      IF (_MessageLevel = E_MessageType.eMessageVerbose)
      THEN
        f_MessageSet(_stMsg);
      END_IF

      _rValue                       := Velocity;
    END_IF
END_CASE
CASE _eState
OF
  E_PROGRESS.READY:
    _fbMoveVelocity[2](
                    Axis            := _AxisRef, 
                    Execute         := TRUE,
                    Velocity        := _rValue, 
                    Acceleration    := Acc, 
                    Deceleration    := Dec, 
                    Jerk            := Jerk, 
                    BufferMode      := BufferMode);

    IF _fbMoveVelocity[2].Error
    THEN
      _eState                       := E_PROGRESS.ERROR;

      _nErrorId                     := _fbMoveVelocity[2].ErrorID;
    
      _stMsg.eType                  := E_MessageType.eMessageError;
      _stMsg.eDevice                := e_Device.Axis + TO_DINT(_AxisRef.NcToPlc.AxisId);
      _stMsg.eSubdevice             :=  e_SubDevice.fbMoveVelocity2;
      _stMsg.iErrorNumber           := _nErrorId;

      _stMsg.sText                  := concat(' : ', TO_STRING(_eState));
    
      f_MessageSet(_stMsg);

    ELSIF (_fbMoveVelocity[2].Busy)
    THEN
      _eState                       := E_PROGRESS.PREPARE;

      _stMsg.eType                  := E_MessageType.eMessageVerbose;
      _stMsg.eDevice                := e_Device.Axis + TO_DINT(_AxisRef.NcToPlc.AxisId);
      _stMsg.eSubdevice             :=  e_SubDevice.fbMoveVelocity2;
      _stMsg.iErrorNumber           := 0;

      _stMsg.sText                  := concat('FB busy: ', TO_STRING(_eState));

      IF (_MessageLevel = E_MessageType.eMessageVerbose)
      THEN
        f_MessageSet(_stMsg);
      END_IF

    ELSIF (_fbMoveVelocity[2].CommandAborted)
    THEN
      _eState                       := E_PROGRESS.PREPARE;

      _stMsg.eType                  := E_MessageType.eMessageError;
      _stMsg.eDevice                := e_Device.Axis + TO_DINT(_AxisRef.NcToPlc.AxisId);
      _stMsg.eSubdevice             :=  e_SubDevice.fbMoveVelocity2;
      _stMsg.iErrorNumber           := 0;

      _stMsg.sText                  := concat('FB aborted: ', TO_STRING(_eState));

      f_MessageSet(_stMsg);

    ELSIF (_fbMoveVelocity[2].InVelocity)
    THEN
      _eState                       := E_PROGRESS.PREPARE;

      _stMsg.eType                  := E_MessageType.eMessageVerbose;
      _stMsg.eDevice                := e_Device.Axis + TO_DINT(_AxisRef.NcToPlc.AxisId);
      _stMsg.eSubdevice             :=  e_SubDevice.fbMoveVelocity2;
      _stMsg.iErrorNumber           := 0;

      _stMsg.sText                  := concat('FB done: ', TO_STRING(_eState));

      IF (_MessageLevel = E_MessageType.eMessageVerbose)
      THEN
        f_MessageSet(_stMsg);
      END_IF
    END_IF
END_CASE
CASE _eState
OF
  E_PROGRESS.WAITING:
    _fbMoveVelocity[2](Axis         := _AxisRef);

    IF _fbMoveVelocity[2].Error
    THEN
      _nErrorId                     := _fbMoveVelocity[2].ErrorID;
    
      _stMsg.eType                  := E_MessageType.eMessageError;
      _stMsg.eDevice                := e_Device.Axis + TO_DINT(_AxisRef.NcToPlc.AxisId);
      _stMsg.eSubdevice             :=  e_SubDevice.fbMoveVelocity2;
      _stMsg.iErrorNumber           := _nErrorId;
    
      _stMsg.sText                  := concat(' : ', TO_STRING(_eState));
  
      f_MessageSet(_stMsg);
    
      _eState                       := E_PROGRESS.ERROR;

    ELSIF (Velocity <> _rValue)
    THEN
      _eState                       := E_PROGRESS.STARTUP;

      _fbMoveVelocity[2](
                    Axis            := _AxisRef, 
                    Execute         := FALSE);

      _stMsg.eType                  := E_MessageType.eMessageVerbose;
      _stMsg.eDevice                := e_Device.Axis + TO_DINT(_AxisRef.NcToPlc.AxisId);
      _stMsg.eSubdevice             :=  e_SubDevice.fbMoveVelocity1;
      _stMsg.iErrorNumber           := 0;

      _stMsg.sText                  := concat('Velocity changed: ', TO_STRING(_rValue));
      _stMsg.sText                  := concat(_stMsg.sText        , ' to ');
      _stMsg.sText                  := concat(_stMsg.sText        , TO_STRING(Velocity));

      IF (_MessageLevel = E_MessageType.eMessageVerbose)
      THEN
        f_MessageSet(_stMsg);
      END_IF

      _rValue                       := Velocity;
    END_IF
END_CASE
CASE _eState
OF
  E_PROGRESS.INIT,
  E_PROGRESS.ERROR:
    _fbMoveVelocity[1](Axis         := _AxisRef,
                       Execute      := FALSE);
    _fbMoveVelocity[2](Axis         := _AxisRef,
                       Execute      := FALSE);
END_CASE


MoveVeloBuffer                      := _eState;
END_METHOD

PROPERTY Override : lreal
GET
Override := _rAxisOverride;
END_GET
SET
_rAxisOverride  := Override;
END_SET
END_PROPERTY

METHOD ReadParameter : E_PROGRESS
VAR_INPUT
  Execute           : BOOL;
  ParameterNumber   : Tc2_MC2.MC_AxisParameter;
END_VAR
VAR_INST
  _eState           : E_PROGRESS;
  _rValue           : LREAL;
  _stMsg            : ST_Message;
END_VAR
IF NOT (__ISVALIDREF(_AxisRef)) THEN  ReadParameter  := E_PROGRESS.ERROR; RETURN; END_IF
IF NOT Execute THEN _eState := E_PROGRESS.INIT; END_IF

CASE _eState
OF
  E_PROGRESS.INIT:
    IF Execute 
    THEN
      memset(ADR(_stMsg),0,SIZEOF(_stMsg));
      _nErrorId                     := 0;
      _rValue                       := 0;
      _eState                       := E_PROGRESS.BUSY;
    END_IF
END_CASE
CASE _eState
OF
  E_PROGRESS.BUSY:
    _eState                         := E_PROGRESS.STARTUP;
    _fbReadParameter(
                    Axis            := _AxisRef, 
                    Enable          := FALSE, 
                    ParameterNumber := ParameterNumber, 
                    ReadMode        := Tc2_MC2.READMODE_ONCE, 
                    Value           => _rValue);
END_CASE
CASE _eState
OF
  E_PROGRESS.STARTUP:
    _eState                         := E_PROGRESS.WAITING;
    _fbReadParameter(
                    Axis            := _AxisRef, 
                    Enable          := TRUE, 
                    ParameterNumber := ParameterNumber, 
                    ReadMode        := Tc2_MC2.READMODE_ONCE, 
                    Value           => _rValue);

    _stMsg.eType                    := E_MessageType.eMessageVerbose;
    _stMsg.eDevice                  := e_Device.Axis + TO_DINT(_AxisRef.NcToPlc.AxisId);
    _stMsg.eSubdevice               := e_SubDevice.fbReadParameter;
    _stMsg.iErrorNumber             := 0;

    _stMsg.sText                    := concat(' : ', TO_STRING(_eState));

    IF (_MessageLevel = E_MessageType.eMessageVerbose)
    THEN
      f_MessageSet(_stMsg);
    END_IF
END_CASE
CASE _eState
OF
  E_PROGRESS.WAITING:
    _fbReadParameter(
                    Axis            := _AxisRef,
                    Value           => _rValue);

    IF (_fbReadParameter.Valid)
    THEN
      _eState                       := E_PROGRESS.WORKING;
      _rValueParameterRead          := _rValue;
    ELSE
      IF (_fbReadParameter.Error)
      THEN
        _eState                     := E_PROGRESS.ERROR;
        _nErrorId                   := _fbReadParameter.ErrorID;

        _stMsg.eType                := E_MessageType.eMessageError;
        _stMsg.eDevice              := e_Device.Axis + TO_DINT(_AxisRef.NcToPlc.AxisId);
        _stMsg.eSubdevice           := e_SubDevice.fbReadParameter;
        _stMsg.iErrorNumber         := _nErrorId;

        _stMsg.sText                := concat(' : ', TO_STRING(_eState));

        f_MessageSet(_stMsg);

        _fbReadParameter(
                    Axis            := _AxisRef, 
                    Enable          := FALSE);
      END_IF
    END_IF
END_CASE
CASE _eState
OF
  E_PROGRESS.WORKING:
    _eState                         := E_PROGRESS.DONE;
    _fbReadParameter(
                    Axis            := _AxisRef, 
                    Enable          := FALSE);

    _stMsg.eType                    := E_MessageType.eMessageVerbose;
    _stMsg.eDevice                  := e_Device.Axis + TO_DINT(_AxisRef.NcToPlc.AxisId);
    _stMsg.eSubdevice               := e_SubDevice.fbReadParameter;
    _stMsg.iErrorNumber             := 0;

    _stMsg.sText                    := concat(' : ', TO_STRING(_eState));

    IF (_MessageLevel = E_MessageType.eMessageVerbose)
    THEN
      f_MessageSet(_stMsg);
    END_IF
END_CASE

ReadParameter                       := _eState;
END_METHOD

PROPERTY ReadParameterValue : LREAL
GET
ReadParameterValue := _rValueParameterRead;
END_GET
END_PROPERTY

METHOD Reset : E_PROGRESS
VAR_INPUT
  Execute           : BOOL;
END_VAR
VAR_INST
  _eState           : E_PROGRESS;
  _rValue           : LREAL;
  _stMsg            : ST_Message;
END_VAR
IF NOT (__ISVALIDREF(_AxisRef)) THEN  Reset  := E_PROGRESS.ERROR; RETURN; END_IF
IF NOT Execute THEN _eState := E_PROGRESS.INIT; END_IF

CASE _eState
OF
  E_PROGRESS.INIT:
    IF Execute 
    THEN
      memset(ADR(_stMsg),0,SIZEOF(_stMsg));
      _nErrorId                   := 0;
      _rValue                     := 0;
      _eState                     := E_PROGRESS.BUSY;
    END_IF
END_CASE
CASE _eState
OF
  E_PROGRESS.BUSY:
    _eState                       := E_PROGRESS.WAITING;
    _fbReset(
              Axis                := _AxisRef, 
              Execute             := FALSE);
END_CASE
CASE _eState
OF
  E_PROGRESS.WAITING:
    _fbReset(
              Axis                := _AxisRef, 
              Execute             := TRUE);

    _AxisRef();

    IF _fbReset.Error
    THEN
      _nErrorId                   := _fbReset.ErrorID;

      _stMsg.eType                := E_MessageType.eMessageError;
      _stMsg.eDevice              := e_Device.Axis + TO_DINT(_AxisRef.NcToPlc.AxisId);
      _stMsg.eSubdevice           := e_SubDevice.fbReset;
      _stMsg.iErrorNumber         := _nErrorId;

      f_MessageSet(_stMsg);
      _fbReset(
              Axis                := _AxisRef, 
              Execute             := FALSE);

      _eState                     := E_PROGRESS.ERROR;
    ELSE
      IF _fbReset.Done OR NOT
         _fbReset.Busy
      THEN
        _eState                   := E_PROGRESS.WORKING;
      END_IF
    END_IF
END_CASE
CASE _eState
OF
  E_PROGRESS.WORKING:
    _eState                       := E_PROGRESS.DONE;
    _fbReset(
              Axis                := _AxisRef, 
              Execute             := FALSE);

    _stMsg.eType                  := E_MessageType.eMessageVerbose;
    _stMsg.eDevice                := e_Device.Axis + TO_DINT(_AxisRef.NcToPlc.AxisId);
    _stMsg.eSubdevice             := e_SubDevice.fbReset;
    _stMsg.iErrorNumber           := 0;

    _stMsg.sText                    := concat(' : ', TO_STRING(_eState));

    IF (_MessageLevel = E_MessageType.eMessageVerbose)
    THEN
      f_MessageSet(_stMsg);
    END_IF
END_CASE


Reset                             := _eState;
END_METHOD

METHOD SendToPos : E_PROGRESS
VAR_INPUT
  Execute         : BOOL;
  Position        : LREAL;
  Vel             : LREAL;
  Acc             : LREAL;
  Dec             : LREAL;
  Jerk            : LREAL;
  BufferMode      : Tc2_MC2.MC_BufferMode;
END_VAR
VAR_INST
  _eState           : E_PROGRESS;
  _rValue           : LREAL;
  _rTarget          : LREAL := 0.5;
  _stMsg            : ST_Message;
END_VAR
IF NOT (__ISVALIDREF(_AxisRef)) THEN  SendToPos  := E_PROGRESS.ERROR; RETURN; END_IF
IF NOT Execute THEN _eState := E_PROGRESS.INIT; END_IF

CASE _eState
OF
  E_PROGRESS.INIT:
    IF Execute 
    THEN
      memset(ADR(_stMsg),0,SIZEOF(_stMsg));
      _nErrorId                     := 0;
      _rValue                       := 0;
      _eState                       := E_PROGRESS.BUSY;

      _stMsg.eType                  := E_MessageType.eMessageVerbose;
      _stMsg.eDevice                := e_Device.Axis + TO_DINT(_AxisRef.NcToPlc.AxisId);
      _stMsg.eSubdevice             := e_SubDevice.fbMoveAbsolute1;
      _stMsg.iErrorNumber           := 0;

      _stMsg.sText                  := concat(' : ', TO_STRING(Position));

      IF (_MessageLevel = E_MessageType.eMessageVerbose)
      THEN
        f_MessageSet(_stMsg);
      END_IF
    END_IF
END_CASE
CASE _eState
OF
  E_PROGRESS.BUSY:
    _eState                         := E_PROGRESS.STARTUP;
    _rValue                         := Position;

    _fbMoveAbsolute[1](Axis         := _AxisRef,
                       Execute      := FALSE);
END_CASE
CASE _eState
OF
  E_PROGRESS.STARTUP:
    _fbMoveAbsolute[1](
                    Axis            := _AxisRef, 
                    Execute         := TRUE,
                    Position        := _rValue, 
                    Velocity        := Vel, 
                    Acceleration    := Acc, 
                    Deceleration    := Dec, 
                    Jerk            := Jerk, 
                    BufferMode      := BufferMode);

    _eState                         := E_PROGRESS.PREPARE;
END_CASE
CASE _eState
OF
  E_PROGRESS.PREPARE:
    _fbMoveAbsolute[1](Axis         := _AxisRef);

    IF (_fbMoveAbsolute[1].Error)
    THEN
      _nErrorId                     := _fbMoveAbsolute[1].ErrorID;
    
      _stMsg.eType                  := E_MessageType.eMessageError;
      _stMsg.eDevice                := e_Device.Axis + TO_DINT(_AxisRef.NcToPlc.AxisId);
      _stMsg.eSubdevice             :=  e_SubDevice.fbMoveAbsolute1;
      _stMsg.iErrorNumber           := _nErrorId;
    
      f_MessageSet(_stMsg);
    
      _eState                         := E_PROGRESS.ERROR;

    ELSIF (_fbMoveAbsolute[1].Active)
    THEN
      _eState                       := E_PROGRESS.WAITING;
    END_IF
END_CASE
CASE _eState
OF
  E_PROGRESS.WAITING:
    _fbMoveAbsolute[1](Axis         := _AxisRef);

    IF (_fbMoveAbsolute[1].Error)
    THEN
      _nErrorId                     := _fbMoveAbsolute[1].ErrorID;
    
      _stMsg.eType                  := E_MessageType.eMessageError;
      _stMsg.eDevice                := e_Device.Axis + TO_DINT(_AxisRef.NcToPlc.AxisId);
      _stMsg.eSubdevice             :=  e_SubDevice.fbMoveAbsolute1;
      _stMsg.iErrorNumber           := _nErrorId;
    
      f_MessageSet(_stMsg);
    
      _eState                         := E_PROGRESS.ERROR;

    ELSIF (_AxisRef.NcToPlc.ActPos > _fbMoveAbsolute[1].Position + _rTarget)
    THEN
      _fbMoveAbsolute[1](Axis       := _AxisRef,
                         Execute    := FALSE);

      _eState                       := E_PROGRESS.DONE;

      _stMsg.eType                  := E_MessageType.eMessageVerbose;
      _stMsg.eDevice                := e_Device.Axis + TO_DINT(_AxisRef.NcToPlc.AxisId);
      _stMsg.eSubdevice             := e_SubDevice.fbMoveAbsolute1;
      _stMsg.iErrorNumber           := 0;

      _stMsg.sText                  := concat(' : ', TO_STRING(_eState));

      IF (_MessageLevel = E_MessageType.eMessageVerbose)
      THEN
        f_MessageSet(_stMsg);
      END_IF
    END_IF
END_CASE

SendToPos                             := _eState;
END_METHOD

METHOD StartUp : E_PROGRESS
VAR_INPUT
  Execute           : BOOL;
END_VAR
VAR_INST
  _eState           : E_PROGRESS;
  _uiEncType        : UDINT;

  _sEncoder,
  _sName            : STRING(30);

  _rValue           : LREAL;
  _stMsg            : ST_Message;
END_VAR
IF NOT (__ISVALIDREF(_AxisRef)) THEN  StartUp  := E_PROGRESS.ERROR; RETURN; END_IF
IF NOT Execute THEN _eState := E_PROGRESS.INIT; END_IF


CASE _eState
OF
  E_PROGRESS.INIT:
    IF Execute 
    THEN
      memset(ADR(_stMsg),0,SIZEOF(_stMsg));
      _nErrorId                     := 0;
      _rValue                       := 0;
      _eState                       := E_PROGRESS.BUSY;
    END_IF
END_CASE
CASE _eState
OF
  E_PROGRESS.BUSY:
    IF (_AxisRef.NcToPlc.AxisId <> 0)
    THEN
      _stMsg.eType                  := E_MessageType.eMessageVerbose;
      _stMsg.eDevice                := e_Device.Axis + TO_DINT(_AxisRef.NcToPlc.AxisId);
      _stMsg.eSubdevice             := e_Subdevice.AxisStartUp;
      _stMsg.iErrorNumber           := 0;
      _stMsg.sText                  := concat('StartUp NcAxisId: ', TO_STRING(_AxisRef.NcToPlc.AxisId));

      IF (_MessageLevel = E_MessageType.eMessageVerbose)
      THEN
        f_MessageSet(_stMsg);
      END_IF

      _eState                       := E_PROGRESS.STARTUP;
    END_IF
END_CASE
CASE _eState
OF
  E_PROGRESS.STARTUP:
    _fbADSRead(
              NETID                 := '', 
              PORT                  := 501, 
              IDXGRP                := (16#5000 + _AxisRef.NcToPlc.AxisId), 
              IDXOFFS               := 16#00000003, // offset for encoder type
              LEN                   := SIZEOF(_nEncoderType), 
              DESTADDR              := ADR(_nEncoderType),
              TMOUT                 := T#200MS,
              READ                  := FALSE);

    // clear required ADS information
    _sAxisName      := _sName       := 'NO NAME';
    _sEncoderType   := _sEncoder    := 'NO TYPE';
    _nEncoderType   := _uiEncType   :=  0;

    _eState                         := E_PROGRESS.PREPARE;
END_CASE
CASE _eState
OF
  E_PROGRESS.PREPARE:
    _fbADSRead(
              NETID                 := '', 
              PORT                  := 501, 
              IDXGRP                := (16#5000 + _AxisRef.NcToPlc.AxisId), 
              IDXOFFS               := 16#00000003, // offset for encoder type
              LEN                   := SIZEOF(_nEncoderType), 
              DESTADDR              := ADR(_nEncoderType),
              TMOUT                 := T#200MS,
              READ                  := TRUE);

    IF (_fbADSRead.ERR)
    THEN
      _nErrorId                     := _fbAdsRead.ERRID;

      _stMsg.eType                  := E_MessageType.eMessageError;
      _stMsg.eDevice                := e_Device.Axis + TO_DINT(_AxisRef.NcToPlc.AxisId);
      _stMsg.eSubdevice             := e_Subdevice.AxisStartUp;
      _stMsg.iErrorNumber           := _nErrorId;
      _stMsg.sText                  := 'StartUp Ads Error Read Encoder Type';

      f_MessageSet(_stMsg);
      _eState                       := E_PROGRESS.ERROR;

    ELSIF (_nEncoderType <> 0)
    THEN
      _uiEncType  := _eEncoderType  := _nEncoderType;
      _sEncoder   := _sEncoderType  := TO_STRING(_eEncoderType);

      _stMsg.eType                  := E_MessageType.eMessageInfo;
      _stMsg.eDevice                := e_Device.Axis + TO_DINT(_AxisRef.NcToPlc.AxisId);
      _stMsg.eSubdevice             := e_Subdevice.AxisStartUp;
      _stMsg.iErrorNumber           := 0;
      _stMsg.sText                  := concat('Encoder Type: ', _sEncoder);

      IF (_MessageLevel < E_MessageType.eMessageError)
      THEN
        f_MessageSet(_stMsg);
      END_IF

      _eState                       := E_PROGRESS.READY;
    END_IF
END_CASE
CASE _eState
OF
  E_PROGRESS.READY:
    _fbADSRead(
            NETID                   := '', 
            PORT                    := 501, 
            IDXGRP                  := (16#4000 + _AxisRef.NcToPlc.AxisId), 
            IDXOFFS                 := 16#00000002, // offset for axis name
            LEN                     := SIZEOF(_sAxisName), 
            DESTADDR                := ADR(_sAxisName),
            READ                    := FALSE);

    _eState                         := E_PROGRESS.WAITING;
END_CASE
CASE _eState
OF
  E_PROGRESS.WAITING:
    _fbADSRead(
            NETID                   := '', 
            PORT                    := 501, 
            IDXGRP                  := (16#4000 + _AxisRef.NcToPlc.AxisId), 
            IDXOFFS                 := 16#00000002, // offset for axis name
            LEN                     := SIZEOF(_sAxisName), 
            DESTADDR                := ADR(_sAxisName),
            READ                    := TRUE);

    IF (_fbADSRead.ERR)
    THEN
      _nErrorId                     := _fbAdsRead.ERRID;

      _stMsg.eType                  := E_MessageType.eMessageError;
      _stMsg.eDevice                := e_Device.Axis + TO_DINT(_AxisRef.NcToPlc.AxisId);;
      _stMsg.eSubdevice             := e_Subdevice.AxisStartUp;
      _stMsg.iErrorNumber           := _nErrorId;
      _stMsg.sText                  := 'StartUp Ads Error Read Axis Name';

      f_MessageSet(_stMsg);
      _eState                       := E_PROGRESS.ERROR;

    ELSIF (_sAxisName <> 'NO NAME')
    THEN
      _sName                        := _sAxisName;

      _stMsg.eType                  := E_MessageType.eMessageInfo;
      _stMsg.eDevice                := e_Device.Axis + TO_DINT(_AxisRef.NcToPlc.AxisId);;
      _stMsg.eSubdevice             := e_Subdevice.AxisStartUp;
      _stMsg.iErrorNumber           := 0;
      _stMsg.sText                  := concat('Axis Name: ', _sName);

      IF (_MessageLevel < E_MessageType.eMessageError)
      THEN
        f_MessageSet(_stMsg);
      END_IF

      _eState                       := E_PROGRESS.WORKING;
    END_IF
END_CASE
CASE _eState
OF
  E_PROGRESS.WORKING:
    _eState                         := E_PROGRESS.DONE;
END_CASE

StartUp                             := _eState;
END_METHOD

METHOD Stop : E_PROGRESS
VAR_INPUT
  Execute           : BOOL;
  Dec               : LREAL;
  Jerk              : LREAL;

END_VAR
VAR_INST
  _eState           : E_PROGRESS;
  _rValue           : LREAL;
  _stMsg            : ST_Message;
END_VAR
IF NOT (__ISVALIDREF(_AxisRef)) THEN  Stop  := E_PROGRESS.ERROR; RETURN; END_IF
IF NOT Execute THEN _eState := E_PROGRESS.INIT; END_IF

CASE _eState
OF
  E_PROGRESS.INIT:
    IF Execute 
    THEN
      memset(ADR(_stMsg),0,SIZEOF(_stMsg));
      _nErrorId                     := 0;
      _rValue                       := 0;
      _eState                       := E_PROGRESS.BUSY;
    END_IF
END_CASE
CASE _eState
OF
  E_PROGRESS.BUSY:
    _eState                         := E_PROGRESS.WAITING;
    _fbStop(
              Axis                  := _AxisRef, 
              Execute               := FALSE, 
              Deceleration          := Dec, 
              Jerk                  := Jerk);
END_CASE
CASE _eState
OF
  E_PROGRESS.WAITING:
    _fbStop(
              Axis                  := _AxisRef, 
              Execute               := TRUE, 
              Deceleration          := Dec, 
              Jerk                  := Jerk);

    IF _fbStop.Error
    THEN
        _nErrorId                   := _fbStop.ErrorID;

        _stMsg.eType                := E_MessageType.eMessageError;
        _stMsg.eDevice              := e_Device.Axis + TO_DINT(_AxisRef.NcToPlc.AxisId);
        _stMsg.eSubdevice           := e_SubDevice.fbStop;
        _stMsg.iErrorNumber         := _nErrorId;

        f_MessageSet(_stMsg);
        _fbStop(
              Axis                  := _AxisRef, 
              Execute               := FALSE);

      _eState                       := E_PROGRESS.ERROR;

    ELSE
      IF _fbStop.Done OR
         _AxisRef.Status.NotMoving
      THEN
        _eState                     := E_PROGRESS.WORKING;

      ELSIF _fbStop.CommandAborted
      THEN
        _eState                     := E_PROGRESS.BUSY;
      END_IF
    END_IF
END_CASE
CASE _eState
OF
  E_PROGRESS.WORKING:
    _fbStop(
              Axis                  := _AxisRef, 
              Execute               := FALSE);

    _eState                         := E_PROGRESS.DONE;
END_CASE


Stop                                := _eState;
END_METHOD

METHOD Template : E_PROGRESS
VAR_INPUT
  Execute           : BOOL;
END_VAR
VAR_INST
  _eState           : E_PROGRESS;
  _rValue           : LREAL;
  _udiErr           : UDINT;
  _stMsg            : ST_Message;


END_VAR
IF NOT (__ISVALIDREF(_AxisRef)) THEN _eState := E_PROGRESS.ERROR; END_IF
IF NOT Execute THEN _eState := E_PROGRESS.INIT; END_IF

CASE _eState
OF
  E_PROGRESS.INIT:
    IF Execute 
    THEN
      memset(ADR(_stMsg),0,SIZEOF(_stMsg));
      _udiErr                       := 0;
      _rValue                       := 0;
      _eState                       := E_PROGRESS.BUSY;
    END_IF
END_CASE
CASE _eState
OF
  E_PROGRESS.BUSY:
    _eState                         := E_PROGRESS.STARTUP;
END_CASE
CASE _eState
OF
  E_PROGRESS.STARTUP:
    _eState                       := E_PROGRESS.PREPARE;
END_CASE
CASE _eState
OF
  E_PROGRESS.PREPARE:
    _eState                         := E_PROGRESS.READY;
END_CASE
CASE _eState
OF
  E_PROGRESS.READY:
    _eState                         := E_PROGRESS.WAITING;
END_CASE
CASE _eState
OF
  E_PROGRESS.WAITING:
    _eState                         := E_PROGRESS.WORKING;
END_CASE
CASE _eState
OF
  E_PROGRESS.WORKING:
    _eState                         := E_PROGRESS.DONE;
END_CASE

Template_1 := _eState;
END_METHOD

METHOD WriteParameter : E_PROGRESS
VAR_INPUT
  Execute           : BOOL;
  Value             : LREAL;
  ParameterNumber   : Tc2_MC2.MC_AxisParameter;
END_VAR
VAR_INST
  _eState           : E_PROGRESS;
  _nParameter       : Tc2_MC2.MC_AxisParameter;
  _rValue           : LREAL;
  _stMsg            : ST_Message;
END_VAR
IF NOT (__ISVALIDREF(_AxisRef)) THEN  WriteParameter  := E_PROGRESS.ERROR; RETURN; END_IF
IF NOT Execute THEN _eState := E_PROGRESS.INIT; END_IF

CASE _eState
OF
  E_PROGRESS.INIT:
    IF Execute 
    THEN
      memset(ADR(_stMsg),0,SIZEOF(_stMsg));
      _nParameter                   := 0;
      _nErrorId                     := 0;
      _rValue                       := 0;
      _eState                       := E_PROGRESS.BUSY;
    END_IF
END_CASE
CASE _eState
OF
  E_PROGRESS.BUSY:
    _eState                         := E_PROGRESS.STARTUP;
    _nParameter                     := ParameterNumber;

    _fbWriteParameter(
                    Axis            := _AxisRef, 
                    Execute         := FALSE, 
                    ParameterNumber := ParameterNumber, 
                    Value           := Value);
END_CASE
CASE _eState
OF
  E_PROGRESS.STARTUP:
    _eState                         := E_PROGRESS.WAITING;
    _fbWriteParameter(
                    Axis            := _AxisRef, 
                    Execute         := TRUE, 
                    ParameterNumber := ParameterNumber, 
                    Value           := Value);

END_CASE
CASE _eState
OF
  E_PROGRESS.WAITING:
    _fbWriteParameter(
                    Axis            := _AxisRef, 
                    ParameterNumber := ParameterNumber, 
                    Value           := Value);

    IF _fbWriteParameter.Error
    THEN
      _nErrorId                     := _fbWriteParameter.ErrorID;

      _stMsg.eType                  := E_MessageType.eMessageError;
      _stMsg.eDevice                := e_Device.Axis + TO_DINT(_AxisRef.NcToPlc.AxisId);
      _stMsg.eSubdevice             := e_SubDevice.fbWriteParameter;
      _stMsg.iErrorNumber           := _nErrorId;

      f_MessageSet(_stMsg);

      _fbWriteParameter(
                    Axis            := _AxisRef,
                    Execute         := FALSE, 
                    ParameterNumber := ParameterNumber, 
                    Value           := Value);


      _eState                       := E_PROGRESS.ERROR;
    ELSE
      IF _fbWriteParameter.Done
      THEN
        _rValue                     := _fbWriteParameter.Value;
        _eState                     := E_PROGRESS.WORKING;
      END_IF
    END_IF

END_CASE
CASE _eState
OF
  E_PROGRESS.WORKING:
    _fbWriteParameter(
                    Axis            := _AxisRef,
                    Execute         := FALSE, 
                    ParameterNumber := ParameterNumber, 
                    Value           := Value);
    _eState                         := E_PROGRESS.DONE;
END_CASE


WriteParameter                      := _eState;
END_METHOD

METHOD WriteParameterPersistent : E_PROGRESS
VAR_INPUT
  Execute           : BOOL;
  Value             : LREAL;
  ParameterNumber   : Tc2_MC2.MC_AxisParameter;
END_VAR
VAR_INST
  _eState           : E_PROGRESS;
  _rValue           : LREAL;
  _stMsg            : ST_Message;
END_VAR
IF NOT (__ISVALIDREF(_AxisRef)) THEN  WriteParameterPersistent  := E_PROGRESS.ERROR; RETURN; END_IF
IF NOT Execute THEN _eState := E_PROGRESS.INIT; END_IF

CASE _eState
OF
  E_PROGRESS.INIT:
    IF Execute 
    THEN
      memset(ADR(_stMsg),0,SIZEOF(_stMsg));
      _nErrorId                     := 0;
      _rValue                       := 0;
      _eState                       := E_PROGRESS.BUSY;
    END_IF
END_CASE
CASE _eState
OF
  E_PROGRESS.BUSY:
    _eState                         := E_PROGRESS.STARTUP;
    _fbWriteParameterPersist(
                    Axis            := _AxisRef, 
                    Execute         := FALSE, 
                    ParameterNumber := ParameterNumber, 
                    Value           := Value);
END_CASE
CASE _eState
OF
  E_PROGRESS.STARTUP:
    _eState                         := E_PROGRESS.WAITING;
    _fbWriteParameterPersist(
                    Axis            := _AxisRef, 
                    Execute         := TRUE, 
                    ParameterNumber := ParameterNumber, 
                    Value           := Value);

END_CASE
CASE _eState
OF
  E_PROGRESS.WAITING:
    _fbWriteParameterPersist(
                    Axis            := _AxisRef, 
                    ParameterNumber := ParameterNumber, 
                    Value           := Value);

    IF (_fbWriteParameterPersist.Error)
    THEN
      _nErrorId                     := _fbWriteParameterPersist.ErrorID;

      _stMsg.eType                  := E_MessageType.eMessageError;
      _stMsg.eDevice                := e_Device.Axis + TO_DINT(_AxisRef.NcToPlc.AxisId);
      _stMsg.eSubdevice             := e_SubDevice.fbWriteParameterPersistent;
      _stMsg.iErrorNumber           := _nErrorId;

      f_MessageSet(_stMsg);

      _fbWriteParameterPersist(
                    Axis            := _AxisRef,
                    Execute         := FALSE, 
                    ParameterNumber := ParameterNumber, 
                    Value           := Value);


      _eState                       := E_PROGRESS.ERROR;
    ELSE
      IF (_fbWriteParameterPersist.Done)
      THEN
        _rValue                     := _fbWriteParameterPersist.Value;
        _eState                     := E_PROGRESS.WORKING;
      END_IF
    END_IF

END_CASE
CASE _eState
OF
  E_PROGRESS.WORKING:
    _fbWriteParameterPersist(
                    Axis            := _AxisRef,
                    Execute         := FALSE, 
                    ParameterNumber := ParameterNumber, 
                    Value           := Value);

    _eState                         := E_PROGRESS.DONE;
END_CASE


WriteParameterPersistent            := _eState;
END_METHOD

END_FUNCTION_BLOCK

// ---- CAM/FB_CamCtrl.TcPOU
FUNCTION_BLOCK FB_CamCtrl EXTENDS FB_CamAxis IMPLEMENTS I_Cam_Ctrl
VAR
  _eInit                    : E_PROGRESS;
  _nAxisIndex               : UINT;       // know thyself

  // get interface from McAxis for access to Reset, Enable, Disable, Halt
  _ItfMcAxis                : ARRAY[1..PLC_CONSTANT.MAX_AXIS] OF I_McAxis;

  // pointers to all; access required for coupling; access by index
  _Axes                     : REFERENCE TO ARRAY[1..PLC_CONSTANT.MAX_AXIS] OF AXIS_REF;

  _Ctrl                     : POINTER TO ARRAY[1..PLC_CONSTANT.MAX_AXIS] OF ST_CAM_CTRL;    // contains command to be executed
  _State                    : POINTER TO ARRAY[1..PLC_CONSTANT.MAX_AXIS] OF ST_CAM_STATE;   // mirrors command with added result

  _Info                     : POINTER TO ARRAY[1..PLC_CONSTANT.MAX_AXIS] OF ST_CAM_INFO;    // Read Camming Info Data
  _Data                     : POINTER TO ARRAY[1..PLC_CONSTANT.MAX_AXIS] OF ST_CAM_DATA;    // Camming parameters

  _MotionFunction           : POINTER TO ARRAY[1..PLC_CONSTANT.MAX_AXIS] OF ST_MOTION_FUNCTION;
  _MotionFunctionPoint      : POINTER TO ARRAY[1..PLC_CONSTANT.MAX_AXIS] OF ST_MOTION_FUNCTION_POINT;

  // local copies of command
  _eCtrl,
  _eCtrlOld                       : E_AXIS_CTRL;

  // execution state
  _eResult                        : E_PROGRESS;   // result of execution state
  _eResultOld                     : E_PROGRESS;   // old result for detecting change
  _eState                         : E_AXIS_STATE; // execution state
END_VAR

PROPERTY Axes : reference TO ARRAY[1..PLC_CONSTANT.MAX_AXIS] OF AXIS_REF
SET
_Axes := Axes;
END_SET
END_PROPERTY

METHOD AxisCamIdle : E_PROGRESS
VAR_INPUT
  Execute           : BOOL;
END_VAR
VAR_INST
  _eResult,
  _eState           : E_PROGRESS;
  _stMsg            : ST_Message;
  _nRetry           : UINT;
END_VAR
IF NOT Execute THEN _eState := E_PROGRESS.INIT; END_IF
IF NOT Check() THEN _eState := E_PROGRESS.ERROR; END_IF

CASE _eState
OF
  E_PROGRESS.INIT:
    IF Execute 
    THEN
      memset(ADR(_stMsg),0,SIZEOF(_stMsg));
      _nRetry                       := 0;
      _eResult                      := _ItfMcAxis[_nAxisIndex].Reset(FALSE);
      _eState                       := E_PROGRESS.BUSY;
    END_IF
END_CASE
CASE _eState
OF
  E_PROGRESS.PREPARE:
    _nRetry                         := _nRetry + 1;
    _eResult                        := _ItfMcAxis[_nAxisIndex].Reset(FALSE);
    _eResult                        := _ItfMcAxis[_nAxisIndex].Enable(FALSE);

    _eState                         := E_PROGRESS.BUSY;

    _stMsg.eType                    := E_MessageType.eMessageInfo;
    _stMsg.eDevice                  := e_Device.Camming + TO_DINT(_AxisSlave.NcToPlc.AxisId);
    _stMsg.eSubdevice               :=  e_SubDevice.fbPowerOn;
    _stMsg.iErrorNumber             := _nErrorId;

    _stMsg.sText                    := concat(TO_STRING(_eCtrl), ' retry: ');
    _stMsg.sText                    := concat(_stMsg.sText, TO_STRING(_nRetry));

    IF (_MessageLevel < E_MessageType.eMessageError)
    THEN
      f_MessageSet(_stMsg);
    END_IF
END_CASE
CASE _eState
OF
  E_PROGRESS.BUSY:
    _eResult                        := _ItfMcAxis[_nAxisIndex].Reset(TRUE);

    IF (_eResult = E_PROGRESS.DONE)
    THEN
      _eState                       := E_PROGRESS.STARTUP;
    END_IF
END_CASE
CASE _eState
OF
  E_PROGRESS.STARTUP:
    _eResult                        := _ItfMcAxis[_nAxisIndex].Reset(FALSE);
    _eResult                        := _ItfMcAxis[_nAxisIndex].Enable(FALSE);
    _eState                         := E_PROGRESS.READY;
END_CASE
CASE _eState
OF
  E_PROGRESS.READY:
    _eResult                        := _ItfMcAxis[_nAxisIndex].Enable(TRUE);

    IF (_nRetry > MAX_RETRY)
    THEN
      _eState                       := E_PROGRESS.ERROR;

    ELSIF (_eResult = E_PROGRESS.DONE)
    THEN
      _ItfMcAxis[_nAxisIndex].Enable(FALSE);
      _eState                       := E_PROGRESS.DONE;

    ELSIF (_eResult = E_PROGRESS.ERROR)
    THEN
      _eState                       := E_PROGRESS.PREPARE;

      _nErrorId                     := _AxisSlave.NcToPlc.ErrorCode;
    
      _stMsg.eType                  := E_MessageType.eMessageError;
      _stMsg.eDevice                := e_Device.Camming + TO_DINT(_AxisSlave.NcToPlc.AxisId);
      _stMsg.eSubdevice             :=  e_SubDevice.fbPowerOn;
      _stMsg.iErrorNumber           := _nErrorId;

      _stMsg.sText                  := concat(TO_STRING(_eCtrl), ' error axis enable: ');
      _stMsg.sText                  := concat(_stMsg.sText, TO_STRING(_nAxisIndex));

      f_MessageSet(_stMsg);
    END_IF
END_CASE

AxisCamIdle                                := _eState;
END_METHOD

METHOD AxisCamIn : E_PROGRESS
VAR_INPUT
  Execute           : BOOL;
END_VAR
VAR_INST
  _eCk              : E_CHECK_STATE;

  _eResult,
  _eState           : E_PROGRESS;
  _rValue           : LREAL;
  _udiErr           : UDINT;
  _stMsg            : ST_Message;

END_VAR
IF NOT Execute THEN _eState := E_PROGRESS.INIT; END_IF
IF NOT Check() THEN _eState := E_PROGRESS.ERROR; END_IF


CASE _eState
OF
  E_PROGRESS.INIT:
    IF Execute 
    THEN
      memset(ADR(_stMsg),0,SIZEOF(_stMsg));
      _udiErr                       := 0;

      IF NOT (_stCamData.nMasterIndex > 0) OR
         NOT (_stCamData.nMasterIndex < PLC_CONSTANT.MAX_AXIS+1)
      THEN
        _eState                     := E_PROGRESS.ERROR;
        _eCk                        := E_CHECK_STATE.CAM_MASTER_AXIS_REF_INVALID;

        _stMsg.eType                := E_MessageType.eMessageError;
        _stMsg.eDevice              := E_Device.Camming + TO_DINT(_AxisSlave.NcToPlc.AxisId);
        _stMsg.eSubdevice           := e_Subdevice.CamControl;
        _stMsg.iErrorNumber         := _stCamData.nMasterIndex;
  
        _stMsg.sText                := concat(' : ', TO_STRING(_eCk));
        f_MessageSet(_stMsg);

      ELSE
        _eState                     := E_PROGRESS.BUSY;
        _eCk                        := E_CHECK_STATE.CHECK_DONE;
        _eResult                    := CamIn(FALSE, _stCamData.nMasterIndex);
      END_IF
    END_IF
END_CASE
CASE _eState
OF
  E_PROGRESS.BUSY:
      _eResult                      := CamIn(TRUE, _stCamData.nMasterIndex);

    IF (_eResult = E_PROGRESS.ERROR)
    THEN
      CamIn(FALSE, _stCamData.nMasterIndex);
      _eState                       := E_PROGRESS.ERROR;
      _udiErr                       := _fbCamInV2.ErrorID;

    ELSIF (_eResult = E_PROGRESS.DONE)
    THEN
      CamIn(FALSE, _stCamData.nMasterIndex);
      _eState                       := E_PROGRESS.DONE;
    END_IF
END_CASE


AxisCamIn                           := _eState;
END_METHOD

METHOD AxisCamInfo : E_PROGRESS
VAR_INPUT
  Execute           : BOOL;
END_VAR
VAR_INST
  _eCk              : E_CHECK_STATE;

  _eResult,
  _eState           : E_PROGRESS;
  _rValue           : LREAL;
  _udiErr           : UDINT;
  _stMsg            : ST_Message;

END_VAR
IF NOT Execute THEN _eState := E_PROGRESS.INIT; END_IF
IF NOT Check() THEN _eState := E_PROGRESS.ERROR; END_IF


CASE _eState
OF
  E_PROGRESS.INIT:
    IF Execute 
    THEN
      memset(ADR(_stMsg),0,SIZEOF(_stMsg));
      _udiErr                       := 0;

      _eState                       := E_PROGRESS.BUSY;
      _eCk                          := E_CHECK_STATE.CHECK_DONE;
      _eResult                      := CamInfo(FALSE, _stCamData.nCamTableId, _stCamData.bAtMasterPosition, _stCamData.rMasterPosition);
    END_IF
END_CASE
CASE _eState
OF
  E_PROGRESS.BUSY:
      _eResult                      := CamInfo(TRUE, _stCamData.nCamTableId, _stCamData.bAtMasterPosition, _stCamData.rMasterPosition);

    IF (_eResult = E_PROGRESS.ERROR)
    THEN
      _eState                       := E_PROGRESS.ERROR;
      CamInfo(FALSE, _stCamData.nCamTableId, _stCamData.bAtMasterPosition, _stCamData.rMasterPosition);

    ELSIF (_eResult = E_PROGRESS.DONE)
    THEN
      _eState                       := E_PROGRESS.READY;
      CamInfo(FALSE, _stCamData.nCamTableId, _stCamData.bAtMasterPosition, _stCamData.rMasterPosition);
    END_IF
END_CASE
CASE _eState
OF
  E_PROGRESS.READY:
    _Info^[_nAxisIndex]             := CamInfoData;

    _stMsg.eType                    := E_MessageType.eMessageInfo;
    _stMsg.eDevice                  := E_Device.Camming + TO_DINT(_AxisSlave.NcToPlc.AxisId);
    _stMsg.eSubdevice               := e_Subdevice.CamControl;
    _stMsg.iErrorNumber             := 0;

    _stMsg.sText                    := concat('CamInfoData : ', TO_STRING(_eState));

    IF (_MessageLevel < E_MessageType.eMessageError)
    THEN
      f_MessageSet(_stMsg);
    END_IF

    _eState                         := E_PROGRESS.DONE;
END_CASE


AxisCamInfo                         := _eState;
END_METHOD

METHOD AxisCamOut : E_PROGRESS
VAR_INPUT
  Execute           : BOOL;
END_VAR
VAR_INST
  _eResult,
  _eState           : E_PROGRESS;
END_VAR
IF NOT Execute THEN _eState := E_PROGRESS.INIT; END_IF
IF NOT Check() THEN _eState := E_PROGRESS.ERROR; END_IF


CASE _eState
OF
  E_PROGRESS.INIT:
    IF Execute 
    THEN
      _eState                       := E_PROGRESS.BUSY;
      _eResult                      := CamOut(FALSE);
    END_IF
END_CASE
CASE _eState
OF
  E_PROGRESS.BUSY:
    _eResult                        := CamOut(TRUE);

    IF (_eResult = E_PROGRESS.ERROR)
    THEN
      CamOut(FALSE);
      _eState                       := E_PROGRESS.ERROR;

    ELSIF (_eResult = E_PROGRESS.DONE)
    THEN
      CamOut(FALSE);
      _eState                       := E_PROGRESS.DONE;
    END_IF
END_CASE


AxisCamOut                          := _eState;
END_METHOD

METHOD AxisCamScaling : E_PROGRESS
VAR_INPUT
  Execute             : BOOL;
END_VAR
VAR_INST
  _eResult,
  _eState             : E_PROGRESS;
  _rValue             : LREAL;
  _udiErr             : UDINT;
  _stMsg              : ST_Message;
END_VAR

IF NOT __ISVALIDREF(_AxisSlave)
THEN
  _eCheck                   := E_CHECK_STATE.CAM_SLAVE_AXIS_REF_INVALID;
  AxisCamScaling            := E_PROGRESS.ERROR;
  RETURN;
END_IF

IF NOT Execute THEN _eState := E_PROGRESS.INIT; END_IF

CASE _eState
OF
  E_PROGRESS.INIT:
    IF Execute 
    THEN
      memset(ADR(_stMsg),0,SIZEOF(_stMsg));
      _udiErr               := 0;
      _rValue               := 0;
      _eState               := E_PROGRESS.BUSY;
      _eResult              := CamScaling(FALSE);
    END_IF
END_CASE
CASE _eState
OF
  E_PROGRESS.BUSY:
    _eResult                := CamScaling(TRUE);
    IF (_eResult = E_PROGRESS.ERROR)
    THEN
      CamScaling(FALSE);
      _eState               := E_PROGRESS.ERROR;

    ELSIF (_eResult = E_PROGRESS.DONE)
    THEN
      CamScaling(FALSE);
      _eState               := E_PROGRESS.DONE;
    END_IF
END_CASE

AxisCamScaling              := _eState;
END_METHOD

PROPERTY AxisCtrl : pointer to ARRAY[1..PLC_CONSTANT.MAX_AXIS] OF st_axis_ctrl
SET
_Ctrl := AxisCtrl;
END_SET
END_PROPERTY

PROPERTY AxisData : pointer to ARRAY[1..PLC_CONSTANT.MAX_AXIS] OF ST_CAM_DATA
SET
_Data := AxisData;
END_SET
END_PROPERTY

PROPERTY AxisIndex : uint
SET
END_SET
END_PROPERTY

PROPERTY AxisInfo : pointer to ARRAY[1..PLC_CONSTANT.MAX_AXIS] OF ST_AXIS_INFO
SET
_Info := AxisInfo;
END_SET
END_PROPERTY

METHOD AxisReadMotionFunction : E_PROGRESS
VAR_INPUT
  Execute             : BOOL;
END_VAR
VAR_INST
  _eResult,
  _eState             : E_PROGRESS;
  _rValue             : LREAL;
  _udiErr             : UDINT;
  _stMsg              : ST_Message;
END_VAR

IF NOT __ISVALIDREF(_AxisSlave)
THEN
  _eCheck                   := E_CHECK_STATE.CAM_SLAVE_AXIS_REF_INVALID;
  AxisReadMotionFunction    := E_PROGRESS.ERROR;
  RETURN;
END_IF

IF NOT Execute THEN _eState := E_PROGRESS.INIT; END_IF

CASE _eState
OF
  E_PROGRESS.INIT:
    IF Execute 
    THEN
      memset(ADR(_stMsg),0,SIZEOF(_stMsg));
      _udiErr               := 0;
      _rValue               := 0;
      _eState               := E_PROGRESS.BUSY;
      _eResult              := ReadMotionFunction(FALSE);
    END_IF
END_CASE
CASE _eState
OF
  E_PROGRESS.BUSY:
    _eResult                := ReadMotionFunction(TRUE);
    IF (_eResult = E_PROGRESS.ERROR)
    THEN
      ReadMotionFunction(FALSE);
      _eState               := E_PROGRESS.ERROR;

    ELSIF (_eResult = E_PROGRESS.DONE)
    THEN
      ReadMotionFunction(FALSE);
      _MotionFunction^[_nAxisIndex]     := ReadMotionFunctionData;
      _eState                           := E_PROGRESS.DONE;
    END_IF
END_CASE

AxisReadMotionFunction      := _eState;
END_METHOD

METHOD AxisReadMotionFunctionPoint : E_PROGRESS
VAR_INPUT
  Execute             : BOOL;
END_VAR
VAR_INST
  _eResult,
  _eState             : E_PROGRESS;
  _rValue             : LREAL;
  _udiErr             : UDINT;
  _stMsg              : ST_Message;
END_VAR

IF NOT __ISVALIDREF(_AxisSlave)
THEN
  _eCheck                       := E_CHECK_STATE.CAM_SLAVE_AXIS_REF_INVALID;
  AxisReadMotionFunctionPoint   := E_PROGRESS.ERROR;
  RETURN;
END_IF

IF NOT Execute THEN _eState := E_PROGRESS.INIT; END_IF

CASE _eState
OF
  E_PROGRESS.INIT:
    IF Execute 
    THEN
      memset(ADR(_stMsg),0,SIZEOF(_stMsg));
      _udiErr               := 0;
      _rValue               := 0;
      _eState               := E_PROGRESS.BUSY;
      _eResult              := ReadMotionFunctionPoint(FALSE);
    END_IF
END_CASE
CASE _eState
OF
  E_PROGRESS.BUSY:
    _eResult                := ReadMotionFunctionPoint(TRUE);
    IF (_eResult = E_PROGRESS.ERROR)
    THEN
      ReadMotionFunctionPoint(FALSE);
      _eState               := E_PROGRESS.ERROR;

    ELSIF (_eResult = E_PROGRESS.DONE)
    THEN
      ReadMotionFunctionPoint(FALSE);
      _MotionFunctionPoint^[_nAxisIndex]  := ReadMotionFunctionPointData;
      _eState                             := E_PROGRESS.DONE;
    END_IF
END_CASE

AxisReadMotionFunctionPoint      := _eState;
END_METHOD

PROPERTY AxisState : pointer to ARRAY[1..PLC_CONSTANT.MAX_AXIS] OF ST_CAM_STATE
SET
_State := AxisState;
END_SET
END_PROPERTY

METHOD AxisWriteMotionFunction : E_PROGRESS
VAR_INPUT
  Execute             : BOOL;
END_VAR
VAR_INST
  _eResult,
  _eState             : E_PROGRESS;
  _rValue             : LREAL;
  _udiErr             : UDINT;
  _stMsg              : ST_Message;
END_VAR

IF NOT __ISVALIDREF(_AxisSlave)
THEN
  _eCheck                       := E_CHECK_STATE.CAM_SLAVE_AXIS_REF_INVALID;
  AxisWriteMotionFunction       := E_PROGRESS.ERROR;
  RETURN;
END_IF

IF NOT Execute THEN _eState := E_PROGRESS.INIT; END_IF

CASE _eState
OF
  E_PROGRESS.INIT:
    IF Execute 
    THEN
      memset(ADR(_stMsg),0,SIZEOF(_stMsg));
      _udiErr               := 0;
      _rValue               := 0;
      _eState               := E_PROGRESS.BUSY;
      _eResult              := WriteMotionFunction(FALSE);
    END_IF
END_CASE
CASE _eState
OF
  E_PROGRESS.BUSY:
    _eResult                := WriteMotionFunction(TRUE);
    IF (_eResult = E_PROGRESS.ERROR)
    THEN
      WriteMotionFunction(FALSE);
      _eState               := E_PROGRESS.ERROR;

    ELSIF (_eResult = E_PROGRESS.DONE)
    THEN
      WriteMotionFunction(FALSE);
      _eState                             := E_PROGRESS.DONE;
    END_IF
END_CASE

AxisWriteMotionFunction     := _eState;
END_METHOD

METHOD AxisWriteMotionFunctionPoint : E_PROGRESS
VAR_INPUT
  Execute             : BOOL;
END_VAR
VAR_INST
  _eResult,
  _eState             : E_PROGRESS;
  _rValue             : LREAL;
  _udiErr             : UDINT;
  _stMsg              : ST_Message;
END_VAR

IF NOT __ISVALIDREF(_AxisSlave)
THEN
  _eCheck                       := E_CHECK_STATE.CAM_SLAVE_AXIS_REF_INVALID;
  AxisWriteMotionFunctionPoint  := E_PROGRESS.ERROR;
  RETURN;
END_IF

IF NOT Execute THEN _eState := E_PROGRESS.INIT; END_IF

CASE _eState
OF
  E_PROGRESS.INIT:
    IF Execute 
    THEN
      memset(ADR(_stMsg),0,SIZEOF(_stMsg));
      _udiErr               := 0;
      _rValue               := 0;
      _eState               := E_PROGRESS.BUSY;
      _eResult              := WriteMotionFunctionPoint(FALSE);
    END_IF
END_CASE
CASE _eState
OF
  E_PROGRESS.BUSY:
    _eResult                := WriteMotionFunctionPoint(TRUE);
    IF (_eResult = E_PROGRESS.ERROR)
    THEN
      WriteMotionFunctionPoint(FALSE);
      _eState               := E_PROGRESS.ERROR;

    ELSIF (_eResult = E_PROGRESS.DONE)
    THEN
      WriteMotionFunctionPoint(FALSE);
      _eState               := E_PROGRESS.DONE;
    END_IF
END_CASE

AxisWriteMotionFunctionPoint := _eState;
END_METHOD

METHOD PRIVATE CamInit : E_PROGRESS
VAR_INPUT
  Execute           : BOOL;
END_VAR
VAR_INST
  _eResult,
  _eState           : E_PROGRESS;
  _rValue           : LREAL;
  _stMsg            : ST_Message;
END_VAR
IF NOT Check() THEN _eState := E_PROGRESS.ERROR; END_IF
IF NOT Execute THEN _eState := E_PROGRESS.INIT; END_IF

CASE _eState
OF
  E_PROGRESS.INIT:
    IF Execute 
    THEN
      memset(ADR(_stMsg),0,SIZEOF(_stMsg));

      _nErrorId                     := 0;
      _rValue                       := 0;
      _eState                       := E_PROGRESS.BUSY;
      _eInit                        := _eState;
    END_IF
END_CASE
CASE _eState
OF
  E_PROGRESS.BUSY:
    _eState                         := E_PROGRESS.STARTUP;
END_CASE
CASE _eState
OF
  E_PROGRESS.STARTUP:
    // keep this for future use
    _eResult                        := E_PROGRESS.DONE;//StartUp(TRUE);
    IF (_eResult = E_PROGRESS.DONE)
    THEN
      _eState                       := E_PROGRESS.PREPARE;
      _ItfMcAxis[_nAxisIndex].Reset(FALSE);
    ELSIF (_eResult = E_PROGRESS.ERROR)
    THEN
      _eState                       := _eResult;

      _stMsg.eType                  := E_MessageType.eMessageError;
      _stMsg.eDevice                := e_Device.Camming + TO_DINT(_AxisSlave.NcToPlc.AxisId);
      _stMsg.eSubdevice             := e_Subdevice.CamStartUp;
      _stMsg.iErrorNumber := _nErrorId  := 6666;

      _stMsg.sText                  := TO_STRING(_eState);
      f_MessageSet(_stMsg);
    END_IF
END_CASE
CASE _eState
OF
  E_PROGRESS.PREPARE:
    _eResult                        := _ItfMcAxis[_nAxisIndex].Reset(TRUE);
    IF (_eResult = E_PROGRESS.DONE)
    THEN
      _eState                       := E_PROGRESS.WORKING;
    ELSIF (_eResult = E_PROGRESS.ERROR)
    THEN
      _eState                       := _eResult;

      _stMsg.eType                  := E_MessageType.eMessageError;
      _stMsg.eDevice                := e_Device.Camming + TO_DINT(_AxisSlave.NcToPlc.AxisId);
      _stMsg.eSubdevice             := e_Subdevice.fbReset;
      _stMsg.iErrorNumber           := _AxisSlave.Status.ErrorID;

      _stMsg.sText                  := TO_STRING(_eState);
      f_MessageSet(_stMsg);
    END_IF
END_CASE
CASE _eState
OF
  E_PROGRESS.READY:
    _eResult                        := _ItfMcAxis[_nAxisIndex].Reset(FALSE);
    _eState                         := E_PROGRESS.WAITING;
END_CASE
CASE _eState
OF
  E_PROGRESS.WAITING:
    _eState                         := E_PROGRESS.WORKING;
END_CASE
CASE _eState
OF
  E_PROGRESS.WORKING:
    _eState                         := E_PROGRESS.DONE;

    _stMsg.eType                    := E_MessageType.eMessageInfo;
    _stMsg.eDevice                  := e_Device.Camming + TO_DINT(_AxisSlave.NcToPlc.AxisId);
    _stMsg.eSubdevice               := e_Subdevice.CamControl;
    _stMsg.iErrorNumber             := 0;
    _stMsg.sText                    := concat('CamInit: ', TO_STRING(_eState));

    IF (_MessageLevel < E_MessageType.eMessageError)
    THEN
      f_MessageSet(_stMsg);
    END_IF
END_CASE

CamInit                            := _eState;
END_METHOD

METHOD PRIVATE Check : BOOL

//-----------------------------------------------------------------------------
IF (_nAxisIndex < 1) OR
   (_nAxisIndex > PLC_CONSTANT.MAX_AXIS)
THEN
  _eCheck                 := E_CHECK_STATE.AXIS_INDEX_OUT_OF_RANGE;
  RETURN;
END_IF
//-----------------------------------------------------------------------------
// get my AXIS_REF pointer for use in base class
//-----------------------------------------------------------------------------
_AxisSlave                := _Axes[_nAxisIndex];
//-----------------------------------------------------------------------------

IF NOT (_ItfMcAxis[_nAxisIndex] <> 0)
THEN
  _eCheck                 := E_CHECK_STATE.CAM_SLAVE_ITF_MC_AXIS_INVALID;
  RETURN;
END_IF


IF NOT (_Ctrl <> 0)
THEN
  _eCheck                 := E_CHECK_STATE.AXIS_CTRL_POINTER_INVALID;
  RETURN;
END_IF

IF NOT (_State <> 0)
THEN
  _eCheck                 := E_CHECK_STATE.AXIS_STATE_POINTER_INVALID;
  RETURN;
END_IF

IF NOT (_Info <> 0)
THEN
  _eCheck                 := E_CHECK_STATE.AXIS_INFO_POINTER_INVALID;
  RETURN;
END_IF

IF NOT (_Data <> 0)
THEN
  _eCheck                 := E_CHECK_STATE.AXIS_DATA_POINTER_INVALID;
  RETURN;
END_IF

IF NOT (_MotionFunction <> 0)
THEN
  _eCheck                 := E_CHECK_STATE.CAM_MOTION_FUNCTION_POINTER_INVALID;
  RETURN;
END_IF

IF NOT (_MotionFunctionPoint <> 0)
THEN
  _eCheck                 := E_CHECK_STATE.CAM_MOTION_FUNCTION_POINT_POINTER_INVALID;
  RETURN;
END_IF


//-----------------------------------------------------------------------------
//  NaN INF check
//-----------------------------------------------------------------------------
IF NOT IsFinite(F_LReal(_Data^[_nAxisIndex].rActivationPosition))
THEN
  _Data^[_nAxisIndex].rActivationPosition               := 0.0;
END_IF

IF NOT IsFinite(F_LReal(_Data^[_nAxisIndex].stCamScalingData.rMasterOffset))
THEN
  _Data^[_nAxisIndex].stCamScalingData.rMasterOffset    := 0.0;
END_IF

IF NOT IsFinite(F_LReal(_Data^[_nAxisIndex].stCamScalingData.rMasterScaling))
THEN
  _Data^[_nAxisIndex].stCamScalingData.rMasterScaling   := 0.0;
END_IF

IF NOT IsFinite(F_LReal(_Data^[_nAxisIndex].stCamScalingData.rSlaveOffset))
THEN
  _Data^[_nAxisIndex].stCamScalingData.rSlaveOffset     := 0.0;
END_IF

IF NOT IsFinite(F_LReal(_Data^[_nAxisIndex].stCamScalingData.rSlaveScaling))
THEN
	_Data^[_nAxisIndex].stCamScalingData.rSlaveScaling   := 0.0;
END_IF
//-----------------------------------------------------------------------------
//-----------------------------------------------------------------------------
_eCheck                   := E_CHECK_STATE.CHECK_DONE;
Check                     := TRUE;
//-----------------------------------------------------------------------------
//-----------------------------------------------------------------------------
END_METHOD

//-------------------------------------------------------------------------------------
//
//  HAUD 2024 01 20
//
//  Cmd
//    - gets state for ctrl
//    - checks for eInit to be done, before any other commands are accepted
//    - prepare your commands here
//    - init what you have to here
//
//-------------------------------------------------------------------------------------
METHOD PRIVATE Cmd  : E_AXIS_STATE
VAR_INPUT
  eCmd              : E_AXIS_CTRL;
END_VAR
VAR_INST
  _IdxMaster        : UINT;
  _stMsg            : ST_Message;
  _estate           : E_AXIS_STATE;
END_VAR
CASE eCmd
OF
  //-------------------------------------------------------------------------------------
  E_AXIS_CTRL.CAM_INIT:
    _eInit    := _eResult             := CamInit(FALSE);
    _estate                           := E_AXIS_STATE.CAM_INIT;
ELSE
  IF (_eInit <> E_PROGRESS.DONE)
  THEN
    _eResult                          := E_PROGRESS.INVALID;
    _estate                           := E_AXIS_STATE.AXIS_NO_INIT;
  ELSE
    CASE eCmd
    OF
      //---------------------------------------------------------------------------------
      E_AXIS_CTRL.AXIS_IDLE:
        _eResult                      := AxisCamIdle(FALSE);
        _estate                       := E_AXIS_STATE.AXIS_IDLE;

      //---------------------------------------------------------------------------------
      E_AXIS_CTRL.CAM_IN:
        _IdxMaster                    := _Data^[_nAxisIndex].nMasterIndex;
        _stCamData                    := _Data^[_nAxisIndex];
        _eResult                      := AxisCamIn(FALSE);
        _estate                       := E_AXIS_STATE.CAM_IN;

      //---------------------------------------------------------------------------------
      E_AXIS_CTRL.CAM_OUT:
        _eResult                      := AxisCamOut(FALSE);
        _estate                       := E_AXIS_STATE.CAM_OUT;

      //---------------------------------------------------------------------------------
      E_AXIS_CTRL.CAM_SCALING:
        _stCamData                    := _Data^[_nAxisIndex];
        _eResult                      := AxisCamScaling(FALSE);
        _eState                       := E_AXIS_STATE.CAM_SCALING;

      //---------------------------------------------------------------------------------
      E_AXIS_CTRL.CAM_INFO:
        _eResult                      := AxisCamInfo(FALSE);
        _estate                       := E_AXIS_STATE.CAM_INFO;

      //---------------------------------------------------------------------------------
      E_AXIS_CTRL.CAM_RD_MOTION_FUNCTION:
        _eResult                      := AxisReadMotionFunction(FALSE);
        _stCamData                    := _Data^[_nAxisIndex];
        _estate                       := E_AXIS_STATE.CAM_RD_MOTION_FUNCTION;

      //---------------------------------------------------------------------------------
      E_AXIS_CTRL.CAM_RD_MOTION_FUNCTION_POINT:
        _eResult                      := AxisReadMotionFunctionPoint(FALSE);
        _stCamData                    := _Data^[_nAxisIndex];
        _estate                       := E_AXIS_STATE.CAM_RD_MOTION_FUNCTION_POINT;

      //---------------------------------------------------------------------------------
      E_AXIS_CTRL.CAM_RD_MOTION_FUNCTIONS_VALUES:
        _stCamData                    := _Data^[_nAxisIndex];
        _estate                       := E_AXIS_STATE.CAM_RD_MOTION_FUNCTIONS_VALUES;

      //---------------------------------------------------------------------------------
      E_AXIS_CTRL.CAM_WRT_MOTION_FUNCTION:
        _eResult                      := AxisWriteMotionFunction(FALSE);
        _stCamData                    := _Data^[_nAxisIndex];
        WriteMotionFunctionData       := _MotionFunction^[_nAxisIndex];
        _estate                       := E_AXIS_STATE.CAM_WRT_MOTION_FUNCTION;

      //---------------------------------------------------------------------------------
      E_AXIS_CTRL.CAM_WRT_MOTION_FUNCTION_POINT:
        _eResult                      := AxisWriteMotionFunctionPoint(FALSE);
        _stCamData                    := _Data^[_nAxisIndex];
        WriteMotionFunctionPointData  := _MotionFunctionPoint^[_nAxisIndex];
        _estate                       := E_AXIS_STATE.CAM_WRT_MOTION_FUNCTION_POINT;

    //-----------------------------------------------------------------------------------
    ELSE
      _estate                         := E_AXIS_STATE.AXIS_NULL;

      IF (eCmd = E_AXIS_CTRL.AXIS_NULL)
      THEN
        _eResult                      := E_PROGRESS.DONE;
      ELSE
        _eResult                      := E_PROGRESS.INVALID;
  
        _stMsg.eType                  := E_MessageType.eMessageError;
        _stMsg.eDevice                := E_Device.Camming + TO_DINT(_AxisSlave.NcToPlc.AxisId);
        _stMsg.eSubdevice             := e_Subdevice.CamControl;
        _stMsg.iErrorNumber           := 0;
  
        _stMsg.sText                  := 'E_AXIS_CTRL.';
        _stMsg.sText                  := concat(_stMsg.sText, TO_STRING(eCmd));
        _stMsg.sText                  := concat(_stMsg.sText, ': ');
        _stMsg.sText                  := concat(_stMsg.sText, TO_STRING(_eResult));

        f_MessageSet(_stMsg);
      END_IF
    END_CASE
  END_IF // _eInit
END_CASE

Cmd                                   := _estate;
END_METHOD

PROPERTY CouplingState : array[0..7] of word
GET
VAR
  wtmp      : ARRAY[0..7] OF WORD;
END_VAR

memcpy(ADR(wtmp[0]) , ADR(_AxisSlave.NcToPlc.CamCouplingState[0]), 1);
memcpy(ADR(wtmp[1]) , ADR(_AxisSlave.NcToPlc.CamCouplingState[1]), 1);
memcpy(ADR(wtmp[2]) , ADR(_AxisSlave.NcToPlc.CamCouplingState[2]), 1);
memcpy(ADR(wtmp[3]) , ADR(_AxisSlave.NcToPlc.CamCouplingState[3]), 1);
memcpy(ADR(wtmp[4]) , ADR(_AxisSlave.NcToPlc.CamCouplingState[4]), 1);
memcpy(ADR(wtmp[5]) , ADR(_AxisSlave.NcToPlc.CamCouplingState[5]), 1);
memcpy(ADR(wtmp[6]) , ADR(_AxisSlave.NcToPlc.CamCouplingState[6]), 1);
memcpy(ADR(wtmp[7]) , ADR(_AxisSlave.NcToPlc.CamCouplingState[7]), 1);

CouplingState := wtmp;
END_GET
END_PROPERTY

METHOD Cycle  : e_progress
VAR_INST
  _eCycle     : E_PROGRESS;

  _eCheckOld  : E_CHECK_STATE;
END_VAR

IF NOT Check() THEN Cycle := _eCycle := _eResult := E_PROGRESS.ERROR; END_IF
//-----------------------------------------------------------------------------
//-----------------------------------------------------------------------------
// OnChange log _eCheck; in case of error --> return to caller
//-----------------------------------------------------------------------------
IF (_eCheck <> _eCheckOld)
THEN
  LogCheck();
  _eCheckOld                        := _eCheck;
END_IF
//-----------------------------------------------------------------------------
IF NOT (_eCheck = E_CHECK_STATE.CHECK_DONE)
THEN
  RETURN;
END_IF
//-----------------------------------------------------------------------------
//-----------------------------------------------------------------------------
// get command from outside world
//-----------------------------------------------------------------------------
_eCtrl                              := _Ctrl^[_nAxisIndex].eCtrl;
//-----------------------------------------------------------------------------
//-----------------------------------------------------------------------------
//  OnChange react to command
//-----------------------------------------------------------------------------
IF (_eCtrl <> _eCtrlOld)
THEN
  // get busy
  _eState                           := Cmd(_eCtrl); // get execution state for command
  _eCtrlOld                         := _eCtrl;
  LogControl();
END_IF
//-----------------------------------------------------------------------------
//-----------------------------------------------------------------------------
//  execution result
//-----------------------------------------------------------------------------
CASE _eResult
OF
  E_PROGRESS.INVALID:
    _State^[_nAxisIndex].eState     := TO_UINT(E_PROGRESS.ERROR);

  E_PROGRESS.ERROR:
    _State^[_nAxisIndex].eState     := _eState + E_PROGRESS.ERROR;

  E_PROGRESS.DONE:
    _State^[_nAxisIndex].eState     := _eState + E_PROGRESS.DONE;

ELSE
    _State^[_nAxisIndex].eState     := _eState + _eResult;
  //-----------------------------------------------------------------------------
  //-----------------------------------------------------------------------------
  //  execution state for command
  //-----------------------------------------------------------------------------
  CASE _eState
  OF
    //---------------------------------------------------------------------------
    E_AXIS_STATE.AXIS_INIT:
      // axis always requires one init from outside world at startup
      // _eInit has to be valid for other commands to be accepted in Cmd(_eCtrl)
      _eInit := _eResult            := CamInit(TRUE);
  
    //---------------------------------------------------------------------------
    E_AXIS_STATE.AXIS_NO_INIT:
      // we are here because you sent a command before having done CAM_INIT
      _eResult                      := E_PROGRESS.ERROR;
  
    //---------------------------------------------------------------------------
    E_AXIS_STATE.AXIS_IDLE:
      _eResult                      := AxisCamIdle(TRUE);
  
    //---------------------------------------------------------------------------
    E_AXIS_STATE.CAM_IN:
      _eResult                      := AxisCamIn(TRUE);
  
    //--------------------------------------------------------------------------
    E_AXIS_STATE.CAM_OUT:
      _eResult                      := AxisCamOut(TRUE);
  
    //--------------------------------------------------------------------------
    E_AXIS_STATE.CAM_SCALING:
      _eResult                      := AxisCamScaling(TRUE);
  
    //--------------------------------------------------------------------------
    E_AXIS_STATE.CAM_INFO:
      _eResult                      := AxisCamInfo(TRUE);
  
    //--------------------------------------------------------------------------
    E_AXIS_STATE.CAM_RD_MOTION_FUNCTION:
      _eResult                      := AxisReadMotionFunction(TRUE);
  
    //--------------------------------------------------------------------------
    E_AXIS_STATE.CAM_RD_MOTION_FUNCTION_POINT:
      _eResult                      := AxisReadMotionFunctionPoint(TRUE);
  
    //--------------------------------------------------------------------------
    E_AXIS_STATE.CAM_WRT_MOTION_FUNCTION:
      _eResult                      := AxisWriteMotionFunction(TRUE);
  
    //--------------------------------------------------------------------------
    E_AXIS_STATE.CAM_WRT_MOTION_FUNCTION_POINT:
      _eResult                      := AxisWriteMotionFunctionPoint(TRUE);
  
  ELSE
    IF (_eCtrl > E_AXIS_CTRL.AXIS_NULL)
    THEN
      _eResult                      := E_PROGRESS.NOT_EXIST;
      _State^[_nAxisIndex].bError   := TRUE;
    ELSE
      _eResult                      := E_PROGRESS.INVALID;
    END_IF
  END_CASE
END_CASE
//-----------------------------------------------------------------------------
//-----------------------------------------------------------------------------
//  OnChange of execution state result
//    - log result and clear error number on interface
//-----------------------------------------------------------------------------
IF (_eResult <> _eResultOld)
THEN
  LogResult();
  _eResultOld                       := _eResult;
END_IF
//-----------------------------------------------------------------------------
//-----------------------------------------------------------------------------
//  CAM couplingstate and TableId freom AXIS_REF
//-----------------------------------------------------------------------------
_State^[_nAxisIndex].wCamCouplingState   := CouplingState;
_State^[_nAxisIndex].nCamCouplingTableId := _AxisSlave.NcToPlc.CamCouplingTableID;
//-----------------------------------------------------------------------------
END_METHOD

PROPERTY ItfMcAxes : array[1..MAX_AXIS] of I_McAxis
SET
_ItfMcAxis := ItfMcAxes;
END_SET
END_PROPERTY

METHOD LogCheck
VAR_INST
  _sChck            : STRING(30);

  _stMsg            : ST_Message;
END_VAR
  _stMsg.eType               := SEL((_eCheck = E_CHECK_STATE.CHECK_DONE),(E_MessageType.eMessageError),(E_MessageType.eMessageInfo));
  _stMsg.eDevice             := E_Device.Camming + TO_DINT(_AxisSlave.NcToPlc.AxisId);
  _stMsg.eSubdevice          := e_Subdevice.CamControl;
  _stMsg.iErrorNumber        := _nAxisIndex;

  _sChck                     := concat('E_CHECK_STATE', '.');
  _sChck                     := concat(_sChck, TO_STRING(_eCheck));

  _stMsg.sText               := concat('cyclic check: ', _sChck);

  IF (_MessageLevel < E_MessageType.eMessageError)
  THEN
    f_MessageSet(_stMsg);
  ELSE
    IF (_stMsg.eType = E_MessageType.eMessageError)
    THEN
      f_MessageSet(_stMsg);
    END_IF
  END_IF
END_METHOD

METHOD PRIVATE LogControl
VAR_INST
  _sResult,
  _sCtrl            : STRING(30);

  _stMsg            : ST_Message;
END_VAR
  _stMsg.eType               := E_MessageType.eMessageInfo;
  _stMsg.eDevice             := E_Device.Camming + TO_DINT(_AxisSlave.NcToPlc.AxisId);
  _stMsg.eSubdevice          := e_Subdevice.CamControl;
  _stMsg.iErrorNumber        := _nAxisIndex;

  _sCtrl                     := concat('E_AXIS_CTRL', '.');
  _sCtrl                     := concat(_sCtrl, TO_STRING(_eCtrl));

  _stMsg.sText               := concat('new command: ', _sCtrl);

  IF (_MessageLevel < E_MessageType.eMessageError)
  THEN
    f_MessageSet(_stMsg);
  ELSE
    IF (_stMsg.eType = E_MessageType.eMessageError)
    THEN
      f_MessageSet(_stMsg);
    END_IF
  END_IF
END_METHOD

METHOD PRIVATE LogResult
VAR_INST
  _sResult,
  _sCtrl            : STRING(30);

  _stMsg            : ST_Message;
END_VAR

  _stMsg.eType               := E_MessageType.eMessageInfo;
  _stMsg.eDevice             := E_Device.Camming + TO_DINT(_AxisSlave.NcToPlc.AxisId);
  _stMsg.eSubdevice          := e_Subdevice.CamControl;
  _stMsg.iErrorNumber        := _nAxisIndex;

  _sCtrl                     := concat('E_AXIS_CTRL', '.');
  _sCtrl                     := concat(_sCtrl, TO_STRING(_eCtrlOld));

  _sResult                   := concat(': E_PROGRESS', '.');
  _sResult                   := concat(_sResult, TO_STRING(_eResult));

  _stMsg.sText               := concat(_sCtrl, ' ');
  _stMsg.sText               := concat(_sCtrl, _sResult);

  IF (_MessageLevel < E_MessageType.eMessageError)
  THEN
    f_MessageSet(_stMsg);
  ELSE
    IF (_stMsg.eType = E_MessageType.eMessageError)
    THEN
      f_MessageSet(_stMsg);
    END_IF
  END_IF
END_METHOD

PROPERTY MotionFunction : POINTER TO ARRAY[1..MAX_AXIS] OF ST_MOTION_FUNCTION
SET
_MotionFunction := MotionFunction;
END_SET
END_PROPERTY

PROPERTY MotionFunctionPoint : pointer to array[1..MAX_AXIS] of ST_MOTION_FUNCTION_POINT
SET
_MotionFunctionPoint := MotionFunctionPoint;
END_SET
END_PROPERTY

END_FUNCTION_BLOCK

// ---- CAM/FB_CamAxis.TcPOU
FUNCTION_BLOCK FB_CamAxis
VAR
  _eCheck                       : E_CHECK_STATE;
  _nErrorId                     : UDINT; // datafield for error

  _MessageLevel                 : E_MessageType;

  _AxisSlave                    : REFERENCE TO AXIS_REF;
  _AxisMaster                   : REFERENCE TO AXIS_REF;

  _fbCamInV2                    : Tc2_MC2_Camming.MC_CamIn_V2;
  _fbScalingV2                  : Tc2_MC2_Camming.MC_CamScaling_V2;
  _fbCamInfoV2                  : Tc2_MC2_Camming.MC_CamInfo_V2;

  _fbCamOut                     : Tc2_MC2_Camming.MC_CamOut;

  _fbSetCamOnlineChangeMode     : Tc2_MC2_Camming.MC_SetCamOnlineChangeMode;

  _fbReadMotionFunction         : Tc2_MC2_Camming.MC_ReadMotionFunction;
  _fbReadMotionFunctionPoint    : Tc2_MC2_Camming.MC_ReadMotionFunctionPoint;
  _fbReadMotionFunctionValues   : Tc2_MC2_Camming.MC_ReadMotionFunctionValues;

  _fbWriteMotionFunction        : Tc2_MC2_Camming.MC_WriteMotionFunction;
  _fbWriteMotionFunctionPoint   : Tc2_MC2_Camming.MC_WriteMotionFunctionPoint;

  _stCamData                    : ST_CAM_DATA;  // camming parameters for function calls

  _mcCamInfoData                : Tc2_MC2_Camming.MC_CamInfoData; // read cam info from NC

  _mcCamRef                     : MC_CAM_REF;
  _mcMotionFunction             : ARRAY[1..MAX_MOTION_FUNCTION_POINTS] OF Tc2_MC2_Camming.MC_MotionFunctionPoint;
  _mcMotionFunctionPoint        : Tc2_MC2_Camming.MC_MotionFunctionPoint;
  _nMotionFunctionSize          : UINT;
END_VAR

METHOD CamIn : E_PROGRESS
VAR_INPUT
  Execute           : BOOL;
  nMasterIndex      : UINT;
END_VAR
VAR_INST
  _eCk              : E_CHECK_STATE;
  _eState           : E_PROGRESS;
  _rValue           : LREAL;
  _udiErr           : UDINT;
  _stMsg            : ST_Message;
END_VAR

IF NOT __ISVALIDREF(_AxisSlave)
THEN
  _eCheck                     := E_CHECK_STATE.CAM_SLAVE_AXIS_REF_INVALID;
  CamIn                       := E_PROGRESS.ERROR;
  RETURN;
END_IF

IF NOT Execute THEN _eState := E_PROGRESS.INIT; END_IF


CASE _eState
OF
  E_PROGRESS.INIT:
    IF Execute 
    THEN
      memset(ADR(_stMsg),0,SIZEOF(_stMsg));
      _udiErr                       := 0;

      IF NOT (nMasterIndex = _stCamData.nMasterIndex)
      THEN
        _eState                     := E_PROGRESS.ERROR;
        _eCk                        := E_CHECK_STATE.CAM_MASTER_AXIS_REF_INVALID;

        _stMsg.eType                := E_MessageType.eMessageError;
        _stMsg.eDevice              := E_Device.Camming + TO_DINT(_AxisSlave.NcToPlc.AxisId);
        _stMsg.eSubdevice           := e_Subdevice.fbCamInV2;
        _stMsg.iErrorNumber         := nMasterIndex;
  
        _stMsg.sText                := concat(' : ', TO_STRING(_eCk));
        f_MessageSet(_stMsg);

      ELSE
        _eState                     := E_PROGRESS.BUSY;
        _eCk                        := E_CHECK_STATE.CHECK_DONE;

        IF (_MessageLevel = E_MessageType.eMessageVerbose)
        THEN
          _stMsg.eType              := E_MessageType.eMessageVerbose;
          _stMsg.eDevice            := E_Device.Camming + TO_DINT(_AxisSlave.NcToPlc.AxisId);
          _stMsg.eSubdevice         := e_Subdevice.fbCamInfoV2;
          _stMsg.iErrorNumber       := 0;
    
          _stMsg.sText              := concat(' : ', TO_STRING(_eState));
          f_MessageSet(_stMsg);
        END_IF

      _fbCamInV2(
          Master                    := _AxisMaster, 
          Slave                     := _AxisSlave, 
          Execute                   := FALSE, 
          ActivationMode            := _stCamData.nActivationMode, 
          ActivationPosition        := _stCamData.rActivationPosition, 
          CamTableID                := _stCamData.nCamTableId,
          Scaling                   := CamScalingData,
          Options                   := CamInOptions);
      END_IF
    END_IF
END_CASE
CASE _eState
OF
  E_PROGRESS.BUSY:
    _fbCamInV2(
          Master                    := _AxisMaster, 
          Slave                     := _AxisSlave, 
          Execute                   := TRUE, 
          ActivationMode            := _stCamData.nActivationMode, 
          ActivationPosition        := _stCamData.rActivationPosition, 
          CamTableID                := _stCamData.nCamTableId);

    IF (_fbCamInV2.Error)
    THEN
      _eState                       := E_PROGRESS.ERROR;
      _udiErr                       := _fbCamInV2.ErrorID;

      _stMsg.eType                  := E_MessageType.eMessageError;
      _stMsg.eDevice                := E_Device.Camming + TO_DINT(_AxisSlave.NcToPlc.AxisId);
      _stMsg.eSubdevice             := e_Subdevice.fbCamInV2;
      _stMsg.iErrorNumber           := _udiErr;

      _stMsg.sText                  := concat(' : ', TO_STRING(_eState));
      f_MessageSet(_stMsg);

      _fbCamInV2(
          Master                    := _AxisMaster, 
          Slave                     := _AxisSlave, 
          Execute                   := FALSE); 

    ELSIF (_fbCamInV2.InSync)
    THEN
      _eState                       := E_PROGRESS.DONE;

      IF (_MessageLevel < E_MessageType.eMessageError)
      THEN
        _stMsg.eType                := E_MessageType.eMessageInfo;
        _stMsg.eDevice              := E_Device.Camming + TO_DINT(_AxisSlave.NcToPlc.AxisId);
        _stMsg.eSubdevice           := e_Subdevice.fbCamInV2;
        _stMsg.iErrorNumber         := 0;
  
        _stMsg.sText                := concat(' : ', TO_STRING(_eState));
        f_MessageSet(_stMsg);
      END_IF

      _fbCamInV2(
          Master                    := _AxisMaster, 
          Slave                     := _AxisSlave, 
          Execute                   := FALSE); 
    END_IF
END_CASE

CamIn                               := _eState;
END_METHOD

METHOD CamInfo : E_PROGRESS
VAR_INPUT
  Execute           : BOOL;
  CamTableID        : Tc2_MC2_Camming.MC_CAM_ID;
  AtMasterPosition  : BOOL;
  MasterPosition    : LREAL;
END_VAR
VAR_INST
  _eState           : E_PROGRESS;
  _rValue           : LREAL;
  _udiErr           : UDINT;
  _stMsg            : ST_Message;
  _stCID            : Tc2_MC2_Camming.MC_CamInfoData;
END_VAR

IF NOT __ISVALIDREF(_AxisSlave)
THEN
  _eCheck                     := E_CHECK_STATE.CAM_SLAVE_AXIS_REF_INVALID;
  CamInfo                     := E_PROGRESS.ERROR;
  RETURN;
END_IF

IF NOT Execute THEN _eState := E_PROGRESS.INIT; END_IF

CASE _eState
OF
  E_PROGRESS.INIT:
    IF Execute 
    THEN
      memset(ADR(_stMsg),0,SIZEOF(_stMsg));
      memset(ADR(_stCID),0,SIZEOF(_stCID));

      _udiErr                       := 0;
      _eState                       := E_PROGRESS.BUSY;

      _fbCamInfoV2(
              Slave                 := _AxisSlave, 
              Execute               := FALSE, 
              CamTableID            := CamTableID, 
              AtMasterPosition      := AtMasterPosition, 
              MasterPosition        := MasterPosition,
              CamInfo               => _mcCamInfoData);

      IF (_MessageLevel = E_MessageType.eMessageVerbose)
      THEN
        _stMsg.eType                := E_MessageType.eMessageVerbose;
        _stMsg.eDevice              := E_Device.Camming + TO_DINT(_AxisSlave.NcToPlc.AxisId);
        _stMsg.eSubdevice           := e_Subdevice.fbCamInfoV2;
        _stMsg.iErrorNumber         := 0;
  
        _stMsg.sText                := concat(' : ', TO_STRING(_eState));
        f_MessageSet(_stMsg);
      END_IF
    END_IF
END_CASE
CASE _eState
OF
  E_PROGRESS.BUSY:
    _fbCamInfoV2(
              Slave                 := _AxisSlave, 
              Execute               := TRUE, 
              CamTableID            := CamTableID, 
              AtMasterPosition      := AtMasterPosition, 
              MasterPosition        := MasterPosition,
              CamInfo               => _mcCamInfoData);

    IF (_fbCamInfoV2.Error)
    THEN
      _eState                       := E_PROGRESS.ERROR;
      _udiErr                       := _fbCamInfoV2.ErrorID;

      _stMsg.eType                  := E_MessageType.eMessageError;
      _stMsg.eDevice                := E_Device.Camming + TO_DINT(_AxisSlave.NcToPlc.AxisId);
      _stMsg.eSubdevice             := e_Subdevice.fbCamInfoV2;
      _stMsg.iErrorNumber           := _udiErr;

      _stMsg.sText                  := concat(' : ', TO_STRING(_eState));
      f_MessageSet(_stMsg);

      _fbCamInfoV2(
              Slave                 := _AxisSlave, 
              Execute               := FALSE);

    ELSIF (_fbCamInfoV2.Done)
    THEN
      _eState                       := E_PROGRESS.DONE;
      _stCID                        := _fbCamInfoV2.CamInfo;

      IF (_MessageLevel < E_MessageType.eMessageError)
      THEN
        _stMsg.eType                := E_MessageType.eMessageInfo;
        _stMsg.eDevice              := E_Device.Camming + TO_DINT(_AxisSlave.NcToPlc.AxisId);
        _stMsg.eSubdevice           := e_Subdevice.fbCamInfoV2;
        _stMsg.iErrorNumber         := 0;
  
        _stMsg.sText                := concat(' : ', TO_STRING(_eState));
        f_MessageSet(_stMsg);
      END_IF
      _fbCamInfoV2(
              Slave                 := _AxisSlave, 
              Execute               := FALSE);
    END_IF
END_CASE

CamInfo                             := _eState;
END_METHOD

PROPERTY CamInfoData : ST_CAM_INFO
GET
VAR
  _stInfoData     : ST_CAM_INFO;
END_VAR


_stInfoData.bPeriodic                       := _mcCamInfoData.Periodic;
_stInfoData.bMasterAbsolute                 := _mcCamInfoData.MasterAbsolute;
_stInfoData.bSlaveAbsolute                  := _mcCamInfoData.SlaveAbsolute;
_stInfoData.bScalingPending                 := _mcCamInfoData.ScalingPending;
_stInfoData.bCamDataQueued                  := _mcCamInfoData.CamDataQueued;
_stInfoData.bCamTableQueued                 := _mcCamInfoData.CamTableQueued;

_stInfoData.nTableType                      := _mcCamInfoData.TableType;
_stInfoData.nInterpolationType              := _mcCamInfoData.InterpolationType;
_stInfoData.nNumberOfRows                   := TO_UINT(_mcCamInfoData.NumberOfRows);
_stInfoData.nNumberOfColumns                := TO_UINT(_mcCamInfoData.NumberOfColumns);
_stInfoData.nMasterAxisId                   := TO_UINT(_mcCamInfoData.MasterAxisId);
_stInfoData.nSlaveAxisId                    := TO_UINT(_mcCamInfoData.SlaveAxisId);

_stInfoData.rMasterCamStartPos              := _mcCamInfoData.MasterCamStartPos;
_stInfoData.rSlaveCamStartPos               := _mcCamInfoData.SlaveCamStartPos;
_stInfoData.rRawMasterPeriod                := _mcCamInfoData.RawMasterPeriod;
_stInfoData.rRawSlaveStroke                 := _mcCamInfoData.RawSlaveStroke;
_stInfoData.rMasterAxisCouplingPos          := _mcCamInfoData.MasterAxisCouplingPos;
_stInfoData.rSlaveAxisCouplingPos           := _mcCamInfoData.SlaveAxisCouplingPos;

_stInfoData.rMasterOffset                   := _mcCamInfoData.MasterOffset;
_stInfoData.rSlaveOffset                    := _mcCamInfoData.SlaveOffset;
_stInfoData.rMasterScaling                  := _mcCamInfoData.MasterScaling;
_stInfoData.rSlaveScaling                   := _mcCamInfoData.SlaveScaling;
_stInfoData.rSumOfSlaveStrokes              := _mcCamInfoData.SumOfSlaveStrokes;
_stInfoData.rSumOfSuperpositionDistance     := _mcCamInfoData.SumOfSuperpositionDistance;
_stInfoData.rActualMasterAxisPos            := _mcCamInfoData.ActualMasterAxisPos;
_stInfoData.rActualSlaveAxisPos             := _mcCamInfoData.ActualSlaveAxisPos;
_stInfoData.rActualMasterCamPos             := _mcCamInfoData.ActualMasterCamPos;
_stInfoData.rActualSlaveCamPos              := _mcCamInfoData.ActualSlaveCamPos;
_stInfoData.rActualPhaseShift               := _mcCamInfoData.ActualPhaseShift;

_stInfoData.nScalingActivationMode          := _mcCamInfoData.ScalingActivationMode;
_stInfoData.rScalingActivationPos           := _mcCamInfoData.ScalingActivationPos;
_stInfoData.nScalingMasterScalingMode       := _mcCamInfoData.ScalingMasterScalingMode;
_stInfoData.nScalingSlaveScalingMode        := _mcCamInfoData.ScalingSlaveScalingMode;

_stInfoData.nOnlineChangeActivationMode     := _mcCamInfoData.OnlineChangeActivationMode;
_stInfoData.rOnlineChangeActivationPos      := _mcCamInfoData.OnlineChangeActivationPos;
_stInfoData.nOnlineChangeMasterScalingMode  := _mcCamInfoData.OnlineChangeMasterScalingMode;
_stInfoData.nOnlineChangeSlaveScalingMode   := _mcCamInfoData.OnlineChangeSlaveScalingMode;

_stInfoData.nCamExchangeCamTableID          := _mcCamInfoData.CamExchangeCamTableID;
_stInfoData.nCamExchangeActivationMode      := _mcCamInfoData.CamExchangeActivationMode;
_stInfoData.rCamExchangeActivationPos       := _mcCamInfoData.CamExchangeActivationPos;
_stInfoData.nCamExchangeMasterScalingMode   := _mcCamInfoData.CamExchangeMasterScalingMode;
_stInfoData.nCamExchangeSlaveScalingMode    := _mcCamInfoData.CamExchangeSlaveScalingMode;
END_GET
END_PROPERTY

PROPERTY CamInOptions : ST_CamInOptions_V2
GET
VAR
  _CamInOptions   : ST_CamInOptions_V2;
END_VAR

_CamInOptions.CamOperationMode      := _stCamData.stOptions.nCamOperationMode;
_CamInOptions.InterpolationType     := _stCamData.stOptions.nInterpolationType;
_CamInOptions.ReferenceCamTableID   := _stCamData.stOptions.nReferenceCamTableId;
END_GET
END_PROPERTY

METHOD CamOut : E_PROGRESS
VAR_INPUT
  Execute           : BOOL;
END_VAR
VAR_INST
  _dwCoupleState    : DWORD;      // debug
  _eState           : E_PROGRESS;
  _rValue           : LREAL;
  _udiErr           : UDINT;
  _stMsg            : ST_Message;
END_VAR

IF NOT __ISVALIDREF(_AxisSlave)
THEN
  _eCheck                     := E_CHECK_STATE.CAM_SLAVE_AXIS_REF_INVALID;
  CamOut                      := E_PROGRESS.ERROR;
  RETURN;
END_IF

IF NOT Execute THEN _eState := E_PROGRESS.INIT; END_IF


CASE _eState
OF
  E_PROGRESS.INIT:
    IF Execute 
    THEN
      memset(ADR(_stMsg),0,SIZEOF(_stMsg));
      _udiErr                       := 0;
      _dwCoupleState                := _AxisSlave.NcToPlc.CoupleState;

      _eState                       := E_PROGRESS.BUSY;

      IF (_MessageLevel = E_MessageType.eMessageVerbose)
      THEN
        _stMsg.eType                := E_MessageType.eMessageInfo;
        _stMsg.eDevice              := E_Device.Camming + TO_DINT(_AxisSlave.NcToPlc.AxisId);
        _stMsg.eSubdevice           := e_Subdevice.fbCamOut;
        _stMsg.iErrorNumber         := 0;
  
        _stMsg.sText                := concat(' : ', TO_STRING(_eState));
        f_MessageSet(_stMsg);
      END_IF
      _fbCamOut(
                Slave               := _AxisSlave, 
                Execute             := FALSE);
    END_IF
END_CASE
CASE _eState
OF
  E_PROGRESS.BUSY:
    _fbCamOut(
              Slave                 := _AxisSlave, 
              Execute               := TRUE);

    IF (_fbCamOut.Error)
    THEN
      _eState                       := E_PROGRESS.ERROR;
      _udiErr                       := _fbCamOut.ErrorID;

      _stMsg.eType                  := E_MessageType.eMessageError;
      _stMsg.eDevice                := E_Device.Camming + TO_DINT(_AxisSlave.NcToPlc.AxisId);
      _stMsg.eSubdevice             := e_Subdevice.fbCamOut;
      _stMsg.iErrorNumber           := _udiErr;

      _stMsg.sText                  := concat(' : ', TO_STRING(_eState));
      f_MessageSet(_stMsg);

      _fbCamOut(
                Slave               := _AxisSlave, 
                Execute             := FALSE);

    ELSIF (_fbCamOut.Done)
    THEN
      _eState                       := E_PROGRESS.DONE;

      IF (_MessageLevel < E_MessageType.eMessageError)
      THEN
        _stMsg.eType                := E_MessageType.eMessageInfo;
        _stMsg.eDevice              := E_Device.Camming + TO_DINT(_AxisSlave.NcToPlc.AxisId);
        _stMsg.eSubdevice           := e_Subdevice.fbCamOut;
        _stMsg.iErrorNumber         := 0;
  
        _stMsg.sText                := concat(' : ', TO_STRING(_eState));
        f_MessageSet(_stMsg);
      END_IF
      _fbCamOut(
                Slave               := _AxisSlave, 
                Execute             := FALSE);
    END_IF
END_CASE

CamOut                              := _eState;
END_METHOD

METHOD CamScaling : E_PROGRESS
VAR_INPUT
  Execute           : BOOL;
END_VAR
VAR_INST
  _eState           : E_PROGRESS;
  _rValue           : LREAL;
  _udiErr           : UDINT;
  _stMsg            : ST_Message;

  _stLastScalingData  : Tc2_MC2_Camming.ST_CamScalingData;
  _nLastCamTableID    : UDINT;
END_VAR

IF NOT __ISVALIDREF(_AxisSlave)
THEN
  _eCheck                     := E_CHECK_STATE.CAM_SLAVE_AXIS_REF_INVALID;
  CamScaling                  := E_PROGRESS.ERROR;
  RETURN;
END_IF

IF NOT Execute THEN _eState   := E_PROGRESS.INIT; END_IF


CASE _eState
OF
  E_PROGRESS.INIT:
    IF Execute 
    THEN
      memset(ADR(_stMsg),0,SIZEOF(_stMsg));
      _udiErr                       := 0;
      _rValue                       := 0;
      _eState                       := E_PROGRESS.BUSY;

      _fbScalingV2(
              Slave                 := _AxisSlave, 
              Execute               := FALSE, 
              ActivationMode        := _stCamData.nActivationMode, 
              ActivationPosition    := _stCamData.rActivationPosition, 
              CamTableID            := _stCamData.nCamTableId,
              Scaling               := CamScalingData);
    END_IF
END_CASE
CASE _eState
OF
  E_PROGRESS.BUSY:
    _eState                         := E_PROGRESS.STARTUP;
    _nLastCamTableID                := _stCamData.nCamTableId;
    _stLastScalingData              := _fbScalingV2.Scaling;

    IF (_MessageLevel = E_MessageType.eMessageVerbose)
    THEN
      _stMsg.eType                  := E_MessageType.eMessageVerbose;
      _stMsg.eDevice                := E_Device.Camming + TO_DINT(_AxisSlave.NcToPlc.AxisId);
      _stMsg.eSubdevice             := e_Subdevice.fbCamScalingV2;
      _stMsg.iErrorNumber           := _nLastCamTableID;

      _stMsg.sText                  := concat(' : ', TO_STRING(_eState));
      f_MessageSet(_stMsg);
    END_IF
END_CASE
CASE _eState
OF
  E_PROGRESS.STARTUP:
      _fbScalingV2(
              Slave                 := _AxisSlave, 
              Execute               := TRUE, 
              ActivationMode        := _stCamData.nActivationMode, 
              ActivationPosition    := _stCamData.rActivationPosition, 
              CamTableID            := _stCamData.nCamTableId);

    IF (_fbScalingV2.Error)
    THEN
      _eState                       := E_PROGRESS.ERROR;
      _udiErr                       := _fbScalingV2.ErrorID;

      _stMsg.eType                  := E_MessageType.eMessageError;
      _stMsg.eDevice                := E_Device.Camming + TO_DINT(_AxisSlave.NcToPlc.AxisId);
      _stMsg.eSubdevice             := e_Subdevice.fbCamScalingV2;
      _stMsg.iErrorNumber           := _udiErr;

      _stMsg.sText                  := concat(' : ', TO_STRING(_eState));
      f_MessageSet(_stMsg);

      _fbScalingV2(
              Slave                 := _AxisSlave, 
              Execute               := FALSE); 

    ELSIF (_fbScalingV2.CommandAborted)
    THEN
      _eState                       := E_PROGRESS.ERROR;
      _udiErr                       := _fbScalingV2.ErrorID;

      _stMsg.eType                  := E_MessageType.eMessageError;
      _stMsg.eDevice                := E_Device.Camming + TO_DINT(_AxisSlave.NcToPlc.AxisId);
      _stMsg.eSubdevice             := e_Subdevice.fbCamScalingV2;
      _stMsg.iErrorNumber           := _udiErr;

      _stMsg.sText                  := concat('command aborted : ', TO_STRING(_eState));
      f_MessageSet(_stMsg);

      _fbScalingV2(
          Slave                     := _AxisSlave, 
          Execute                   := FALSE); 

    ELSIF (_fbScalingV2.Done)
    THEN
      _eState                       := E_PROGRESS.DONE;

      IF (_MessageLevel < E_MessageType.eMessageError)
      THEN
        _stMsg.eType                := E_MessageType.eMessageInfo;
        _stMsg.eDevice              := E_Device.Camming + TO_DINT(_AxisSlave.NcToPlc.AxisId);
        _stMsg.eSubdevice           := e_Subdevice.fbCamScalingV2;
        _stMsg.iErrorNumber         := 0;
  
        _stMsg.sText                := concat(' : ', TO_STRING(_eState));
        f_MessageSet(_stMsg);
      END_IF
      _fbScalingV2(
              Slave                 := _AxisSlave, 
              Execute               := FALSE); 
    END_IF
END_CASE

CamScaling                          := _eState;
END_METHOD

PROPERTY CamScalingData : Tc2_MC2_Camming.ST_CamScalingData
GET
VAR
 _ScaleData   : Tc2_MC2_Camming.ST_CamScalingData;
END_VAR

_ScaleData.MasterOffset       := _stCamData.stCamScalingData.rMasterOffset;
_ScaleData.MasterRelative     := _stCamData.stCamScalingData.bMasterRelative;
_ScaleData.MasterScaling      := _stCamData.stCamScalingData.rMasterScaling;
_ScaleData.MasterScalingMode  := _stCamData.stCamScalingData.nMasterScalingMode;

_ScaleData.SlaveOffset        := _stCamData.stCamScalingData.rSlaveOffset;
_ScaleData.SlaveRelative      := _stCamData.stCamScalingData.bSlaveRelative;
_ScaleData.SlaveScaling       := _stCamData.stCamScalingData.rSlaveScaling;
_ScaleData.SlaveScalingMode   := _stCamData.stCamScalingData.nSlaveScalingMode;

CamScalingData                := _ScaleData;
END_GET
END_PROPERTY

PROPERTY MessageLevel : E_MessageType
SET
_MessageLevel := MessageLevel;
END_SET
END_PROPERTY

METHOD ReadMotionFunction : E_PROGRESS
VAR_INPUT
  Execute           : BOOL;
END_VAR
VAR_INST
  _eState           : E_PROGRESS;
  _rValue           : LREAL;
  _udiErr           : UDINT;
  _stMsg            : ST_Message;


  _nNumPointsRead   : UINT;
END_VAR

IF NOT Execute THEN _eState   := E_PROGRESS.INIT; END_IF


CASE _eState
OF
  E_PROGRESS.INIT:
    IF Execute 
    THEN
      memset(ADR(_mcMotionFunction),0,SIZEOF(_mcMotionFunction));
      memset(ADR(_stMsg),0,SIZEOF(_stMsg));
      _nNumPointsRead               := 0;
      _udiErr                       := 0;
      _rValue                       := 0;
      _eState                       := E_PROGRESS.BUSY;

      _mcCamRef.pArray              := ADR(_mcMotionFunction);
      _mcCamRef.ArraySize           := SIZEOF(_mcMotionFunction);

      _mcCamRef.TableType           := Tc2_MC2_Camming.MC_TABLETYPE_MOTIONFUNCTION;
      _mcCamRef.NoOfColumns         := 1;

      _fbReadMotionFunction(
              Execute               := FALSE, 
              CamTableID            := _stCamData.nCamTableId, 
              PointID               := _stCamData.nPointId,     // must be greater 0
              NumPoints             := _stCamData.nNumPoints,   // 0 = read all
              CamTable              := _mcCamRef);

    END_IF
END_CASE
CASE _eState
OF
  E_PROGRESS.BUSY:
    _fbReadMotionFunction(
              Execute               := TRUE, 
              CamTableID            := _stCamData.nCamTableId,  // ID of the loaded table
              PointID               := _stCamData.nPointId,     // Point ID of the first point to be read
              NumPoints             := _stCamData.nNumPoints,   // 0 = read all points
              CamTable              := _mcCamRef);

    IF (_fbReadMotionFunction.Error)
    THEN
      _eState                       := E_PROGRESS.ERROR;
      _udiErr                       := _fbReadMotionFunction.ErrorID;

      _stMsg.eType                  := E_MessageType.eMessageError;
      _stMsg.eDevice                := E_Device.Camming + TO_DINT(_AxisSlave.NcToPlc.AxisId);
      _stMsg.eSubdevice             := e_Subdevice.fbReadMotionFunction;
      _stMsg.iErrorNumber           := _udiErr;

      _stMsg.sText                  := concat(' : ', TO_STRING(_eState));
      f_MessageSet(_stMsg);

      _fbReadMotionFunction(
              Execute               := FALSE, 
              CamTableID            := _stCamData.nCamTableId,  // ID of the loaded table
              PointID               := _stCamData.nPointId,     // Point ID of the first point to be read
              NumPoints             := _stCamData.nNumPoints,   // 0 = read all points
              CamTable              := _mcCamRef);

    ELSIF (_fbReadMotionFunction.Done)
    THEN
      _eState                       := E_PROGRESS.WORKING;

      IF (_MessageLevel < E_MessageType.eMessageError)
      THEN
        _stMsg.eType                := E_MessageType.eMessageInfo;
        _stMsg.eDevice              := E_Device.Camming + TO_DINT(_AxisSlave.NcToPlc.AxisId);
        _stMsg.eSubdevice           := e_Subdevice.fbReadMotionFunction;
        _stMsg.iErrorNumber         := 0;
  
        _stMsg.sText                := concat(' : ', TO_STRING(_eState));
        f_MessageSet(_stMsg);
      END_IF
    END_IF
END_CASE
CASE _eState
OF
  E_PROGRESS.WORKING:
    _eState                         := E_PROGRESS.FINISHING;
    _nNumPointsRead                 := TO_UINT(_fbReadMotionFunction.NumPointsRead);
    _nMotionFunctionSize            := SEL((TO_UINT(_mcCamRef.ArraySize) > MAX_MOTION_FUNCTION_POINTS),
                                            TO_UINT(_mcCamRef.ArraySize),
                                            MAX_MOTION_FUNCTION_POINTS);

    memcpy(ADR(_mcMotionFunction), _mcCamRef.pArray, _nMotionFunctionSize); 

    _stMsg.eType                    := SEL((TO_UINT(_mcCamRef.ArraySize) > MAX_MOTION_FUNCTION_POINTS),
                                            E_MessageType.eMessageInfo,
                                            E_MessageType.eMessageWarn);

    _stMsg.eDevice                  := E_Device.Camming + TO_DINT(_AxisSlave.NcToPlc.AxisId);
    _stMsg.eSubdevice               := e_Subdevice.fbReadMotionFunction;
    _stMsg.iErrorNumber             := _nMotionFunctionSize;

    _stMsg.sText                    := concat(' : ', TO_STRING(_eState));

    IF (_MessageLevel < E_MessageType.eMessageError)
    THEN
      f_MessageSet(_stMsg);
    END_IF

END_CASE
CASE _eState
OF
  E_PROGRESS.FINISHING:
    _eState                         := E_PROGRESS.DONE;

(*
    _stMotionFunction.stMotionFunction    := _mcMotionFunction;
    _stMotionFunction.nMotionFunctionSize := _nMotionFunctionSize;
    _stMotionFunction.nPoints             := TO_UINT(_fbReadMotionFunction.NumPointsRead);
*)

    IF (_MessageLevel < E_MessageType.eMessageError)
    THEN
      _stMsg.eType                  := E_MessageType.eMessageInfo;
      _stMsg.eDevice                := E_Device.Camming + TO_DINT(_AxisSlave.NcToPlc.AxisId);
      _stMsg.eSubdevice             := e_Subdevice.fbReadMotionFunction;
      _stMsg.iErrorNumber           := 0;
  
      _stMsg.sText                  := concat(' : ', TO_STRING(_eState));
      f_MessageSet(_stMsg);
    END_IF

    _fbReadMotionFunction(
              Execute               := FALSE, 
              CamTableID            := _stCamData.nCamTableId, 
              PointID               := _stCamData.nPointId, 
              NumPoints             := _stCamData.nNumPoints, 
              CamTable              := _mcCamRef);
END_CASE

ReadMotionFunction                  := _eState;
END_METHOD

PROPERTY ReadMotionFunctionData : ST_MOTION_FUNCTION
GET
VAR
  _idx        : UINT;
  _stMf       : ST_MOTION_FUNCTION;
END_VAR

_stMf.nMotionFunctionSize   := TO_UINT(_mcCamRef.ArraySize);
_stMf.nPoints               := TO_UINT(_mcCamRef.NoOfRows);

FOR _idx := 1 TO MAX_MOTION_FUNCTION_POINTS
DO
  IF NOT (_idx > _stMf.nPoints)
  THEN
    _stMf.stMotionFunction[_idx].nFunctionType      := TO_UINT(_mcMotionFunction[_idx].FunctionType);
    _stMf.stMotionFunction[_idx].nPointIndex        := TO_UINT(_mcMotionFunction[_idx].PointIndex);
    _stMf.stMotionFunction[_idx].nRelIndexNextPoint := TO_UINT(_mcMotionFunction[_idx].RelIndexNextPoint);

    _stMf.stMotionFunction[_idx].wPointType         := TO_WORD(_mcMotionFunction[_idx].PointType);

    _stMf.stMotionFunction[_idx].rMasterPos         := _mcMotionFunction[_idx].MasterPos;
    _stMf.stMotionFunction[_idx].rSlavePos          := _mcMotionFunction[_idx].SlavePos;

    _stMf.stMotionFunction[_idx].rSlaveVelo         := _mcMotionFunction[_idx].SlaveVelo;
    _stMf.stMotionFunction[_idx].rSlaveAcc          := _mcMotionFunction[_idx].SlaveAcc;
    _stMf.stMotionFunction[_idx].rSlaveJerk         := _mcMotionFunction[_idx].SlaveJerk;
  END_IF
END_FOR

ReadMotionFunctionData := _stMf;
END_GET
END_PROPERTY

METHOD ReadMotionFunctionPoint : E_PROGRESS
VAR_INPUT
  Execute           : BOOL;
END_VAR
VAR_INST
  _eState           : E_PROGRESS;
  _rValue           : LREAL;
  _udiErr           : UDINT;
  _stMsg            : ST_Message;
END_VAR

IF NOT Execute THEN _eState   := E_PROGRESS.INIT; END_IF


CASE _eState
OF
  E_PROGRESS.INIT:
    IF Execute 
    THEN
      memset(ADR(_mcMotionFunctionPoint),0,SIZEOF(_mcMotionFunctionPoint));
      memset(ADR(_stMsg),0,SIZEOF(_stMsg));
      _udiErr                       := 0;
      _rValue                       := 0;
      _eState                       := E_PROGRESS.BUSY;

      _fbReadMotionFunctionPoint(
              Execute               := FALSE, 
              CamTableID            := _stCamData.nCamTableId, 
              PointID               := _stCamData.nPointId,
              Point                 := _mcMotionFunctionPoint);
    END_IF
END_CASE
CASE _eState
OF
  E_PROGRESS.BUSY:
    _fbReadMotionFunctionPoint(
              Execute               := TRUE, 
              CamTableID            := _stCamData.nCamTableId, 
              PointID               := _stCamData.nPointId,
              Point                 := _mcMotionFunctionPoint);

    IF (_fbReadMotionFunctionPoint.Error)
    THEN
      _eState                       := E_PROGRESS.ERROR;
      _udiErr                       := _fbReadMotionFunctionPoint.ErrorID;

      _stMsg.eType                  := E_MessageType.eMessageError;
      _stMsg.eDevice                := E_Device.Camming + TO_DINT(_AxisSlave.NcToPlc.AxisId);
      _stMsg.eSubdevice             := e_Subdevice.fbReadMotionFunctionPoint;
      _stMsg.iErrorNumber           := _udiErr;

      _stMsg.sText                  := concat(' : ', TO_STRING(_eState));
      f_MessageSet(_stMsg);

      _fbReadMotionFunctionPoint(
              Execute               := FALSE, 
              CamTableID            := _stCamData.nCamTableId, 
              PointID               := _stCamData.nPointId,
              Point                 := _mcMotionFunctionPoint);
    ELSE
      IF (_fbReadMotionFunctionPoint.Done)
      THEN
        _eState                     := E_PROGRESS.DONE;
  
        _stMsg.eType                := E_MessageType.eMessageInfo;
        _stMsg.eDevice              := E_Device.Camming + TO_DINT(_AxisSlave.NcToPlc.AxisId);
        _stMsg.eSubdevice           := e_Subdevice.fbReadMotionFunctionPoint;
        _stMsg.iErrorNumber         := 0;
  
        _stMsg.sText                := concat(' : ', TO_STRING(_eState));

        IF (_MessageLevel < E_MessageType.eMessageError)
        THEN
          f_MessageSet(_stMsg);
        END_IF

        _fbReadMotionFunctionPoint(
              Execute               := FALSE, 
              CamTableID            := _stCamData.nCamTableId, 
              PointID               := _stCamData.nPointId,
              Point                 := _mcMotionFunctionPoint);
      END_IF
    END_IF
END_CASE

ReadMotionFunctionPoint             := _eState;
END_METHOD

PROPERTY ReadMotionFunctionPointData : ST_MOTION_FUNCTION_POINT
GET
VAR
  _stTmp    : ST_MOTION_FUNCTION_POINT;
END_VAR

_stTmp.nFunctionType        := TO_UINT(_mcMotionFunctionPoint.FunctionType);
_stTmp.nPointIndex          := TO_UINT(_mcMotionFunctionPoint.PointIndex);
_stTmp.nRelIndexNextPoint   := TO_UINT(_mcMotionFunctionPoint.RelIndexNextPoint);
_stTmp.wPointType           := TO_WORD(_mcMotionFunctionPoint.PointType);

